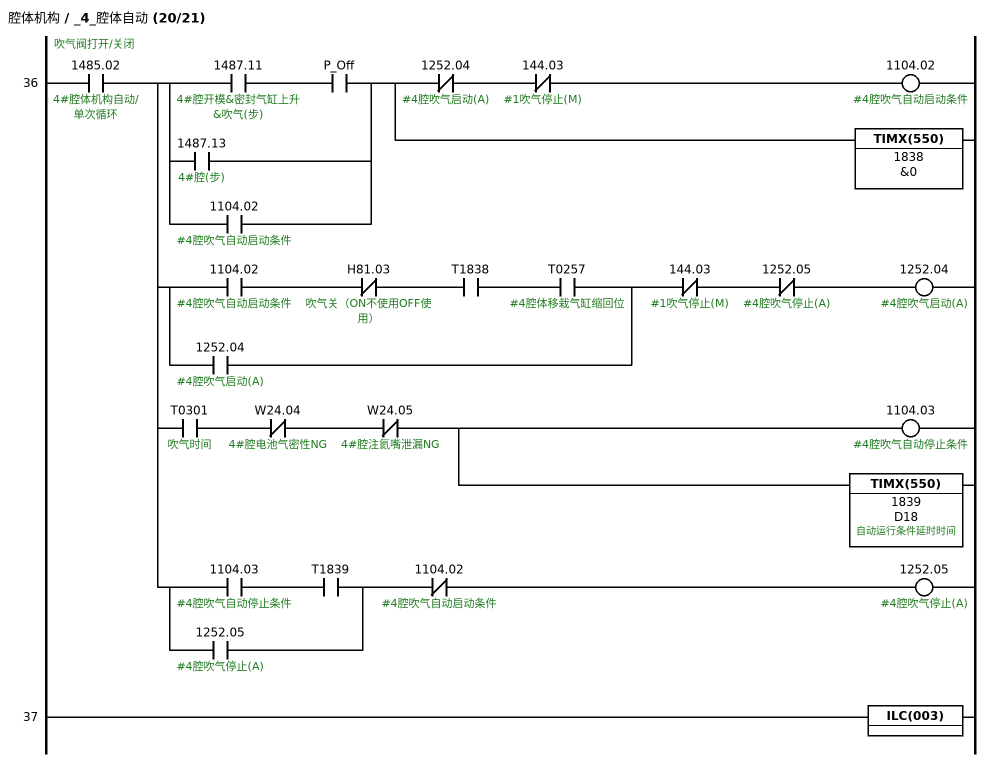
; [picture p360: 腔体机构 / _4_腔体自动, rungs 36-37]
; rung 36: 吹气阀打开/关闭
LD 1485.02  ; 4#腔体机构自动/单次循环
OUT TR0
LD 1487.11  ; 4#腔开模&密封气缸上升&吹气(步)
AND P_Off
OR 1487.13  ; 4#腔(步)
OR 1104.02  ; #4腔吹气自动启动条件
ANDLD
OUT TR1
ANDNOT 1252.04  ; #4腔吹气启动(A)
ANDNOT 144.03  ; #1吹气停止(M)
OUT 1104.02  ; #4腔吹气自动启动条件
LD TR1
TIMX(550) 1838 &0
LD TR0
LD 1104.02  ; #4腔吹气自动启动条件
ANDNOT H81.03  ; 吹气关（ON不使用OFF使用）
AND T1838
AND T0257  ; #4腔体移栽气缸缩回位
OR 1252.04  ; #4腔吹气启动(A)
ANDLD
ANDNOT 144.03  ; #1吹气停止(M)
ANDNOT 1252.05  ; #4腔吹气停止(A)
OUT 1252.04  ; #4腔吹气启动(A)
LD TR0
AND T0301  ; 吹气时间
ANDNOT W24.04  ; 4#腔电池气密性NG
ANDNOT W24.05  ; 4#腔注氦嘴泄漏NG
OUT 1104.03  ; #4腔吹气自动停止条件
TIMX(550) 1839 D18  ; 自动运行条件延时时间
LD TR0
LD 1104.03  ; #4腔吹气自动停止条件
AND T1839
OR 1252.05  ; #4腔吹气停止(A)
ANDLD
ANDNOT 1104.02  ; #4腔吹气自动启动条件
OUT 1252.05  ; #4腔吹气停止(A)
; rung 37
ILC(003)

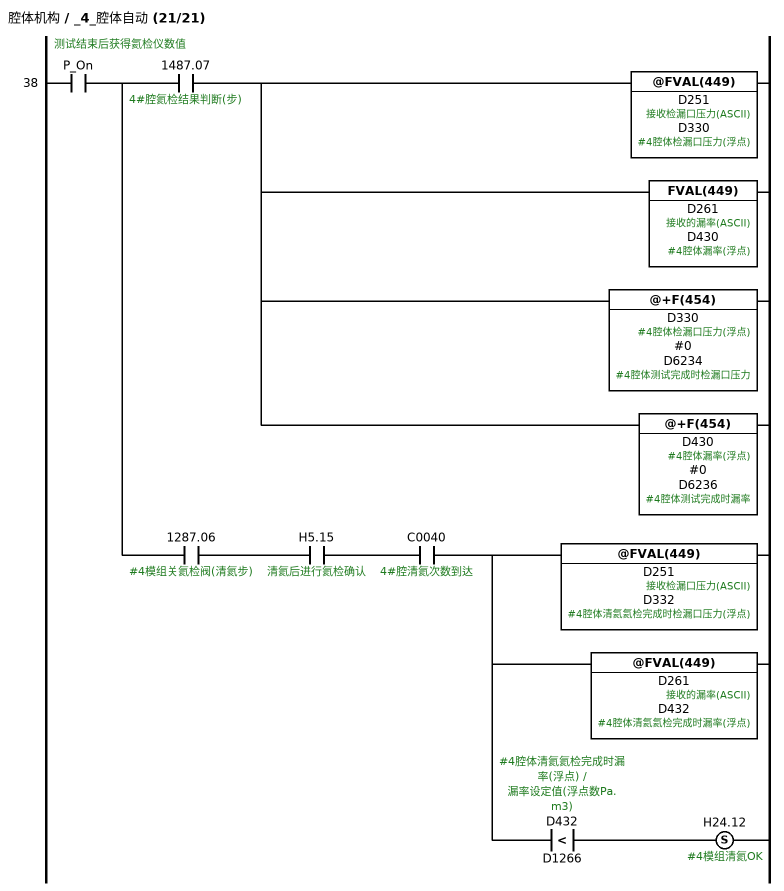
; rung 38: 测试结束后获得氦检仪数值
LD P_On
OUT TR0
AND 1487.07  ; 4#腔氦检结果判断(步)
@FVAL(449) D251 D330  ; 接收检漏口压力(ASCII), #4腔体检漏口压力(浮点)
FVAL(449) D261 D430  ; 接收的漏率(ASCII), #4腔体漏率(浮点)
@+F(454) D330 #0 D6234  ; #4腔体检漏口压力(浮点), #4腔体测试完成时检漏口压力
@+F(454) D430 #0 D6236  ; #4腔体漏率(浮点), #4腔体测试完成时漏率
LD TR0
AND 1287.06  ; #4模组关氦检阀(清氦步)
AND H5.15  ; 清氦后进行氦检确认
AND C0040  ; 4#腔清氦次数到达
@FVAL(449) D251 D332  ; 接收检漏口压力(ASCII), #4腔体清氦氦检完成时检漏口压力(浮点)
@FVAL(449) D261 D432  ; 接收的漏率(ASCII), #4腔体清氦氦检完成时漏率(浮点)
AND<F(331) D432 D1266  ; #4腔体清氦氦检完成时漏率(浮点), 漏率设定值(浮点数Pa.m3)
SET H24.12  ; #4模组清氦OK

### Section 外部输出

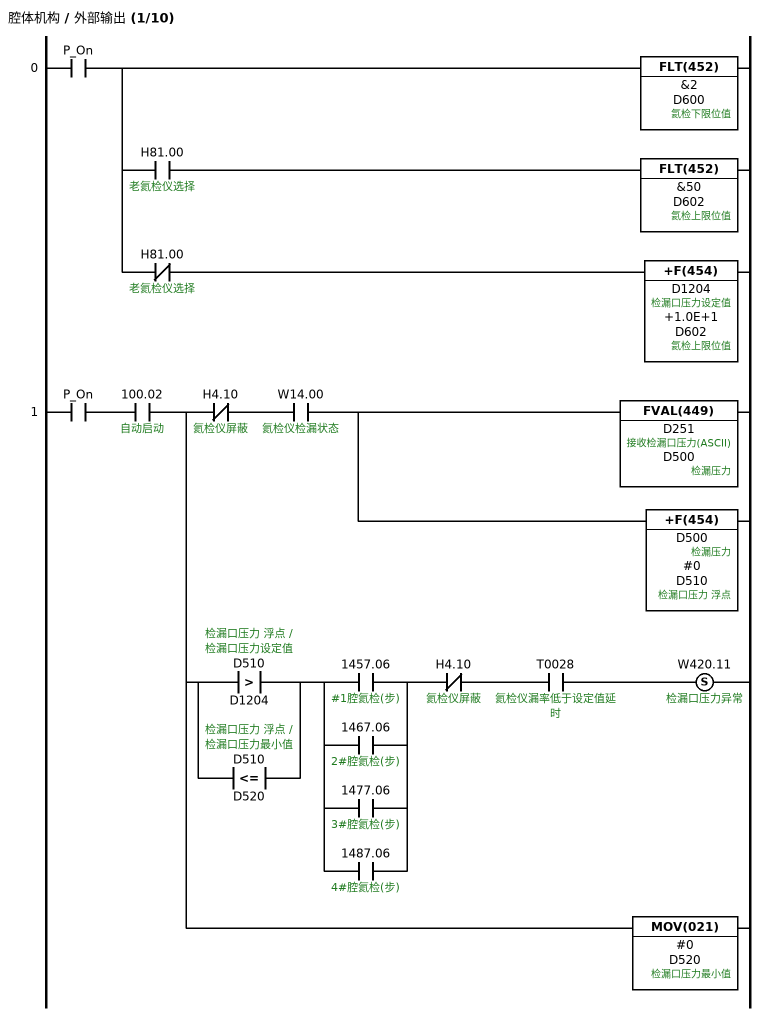
; rung 0
LD P_On
OUT TR0
FLT(452) &2 D600  ; 氦检下限位值
AND H81.00  ; 老氦检仪选择
FLT(452) &50 D602  ; 氦检上限位值
LD TR0
ANDNOT H81.00  ; 老氦检仪选择
+F(454) D1204 +1.0E+1 D602  ; 检漏口压力设定值, 氦检上限位值
; rung 1
LD P_On
AND 100.02  ; 自动启动
OUT TR0
ANDNOT H4.10  ; 氦检仪屏蔽
AND W14.00  ; 氦检仪检漏状态
FVAL(449) D251 D500  ; 接收检漏口压力(ASCII), 检漏压力
+F(454) D500 #0 D510  ; 检漏压力, 检漏口压力 浮点
LD TR0
LD>F(333) D510 D1204  ; 检漏口压力 浮点, 检漏口压力设定值
OR<=F(332) D510 D520  ; 检漏口压力 浮点, 检漏口压力最小值
ANDLD
LD 1457.06  ; #1腔氦检(步)
OR 1467.06  ; 2#腔氦检(步)
OR 1477.06  ; 3#腔氦检(步)
OR 1487.06  ; 4#腔氦检(步)
ANDLD
ANDNOT H4.10  ; 氦检仪屏蔽
AND T0028  ; 氦检仪漏率低于设定值延时
SET W420.11  ; 检漏口压力异常
LD TR0
MOV(021) #0 D520  ; 检漏口压力最小值

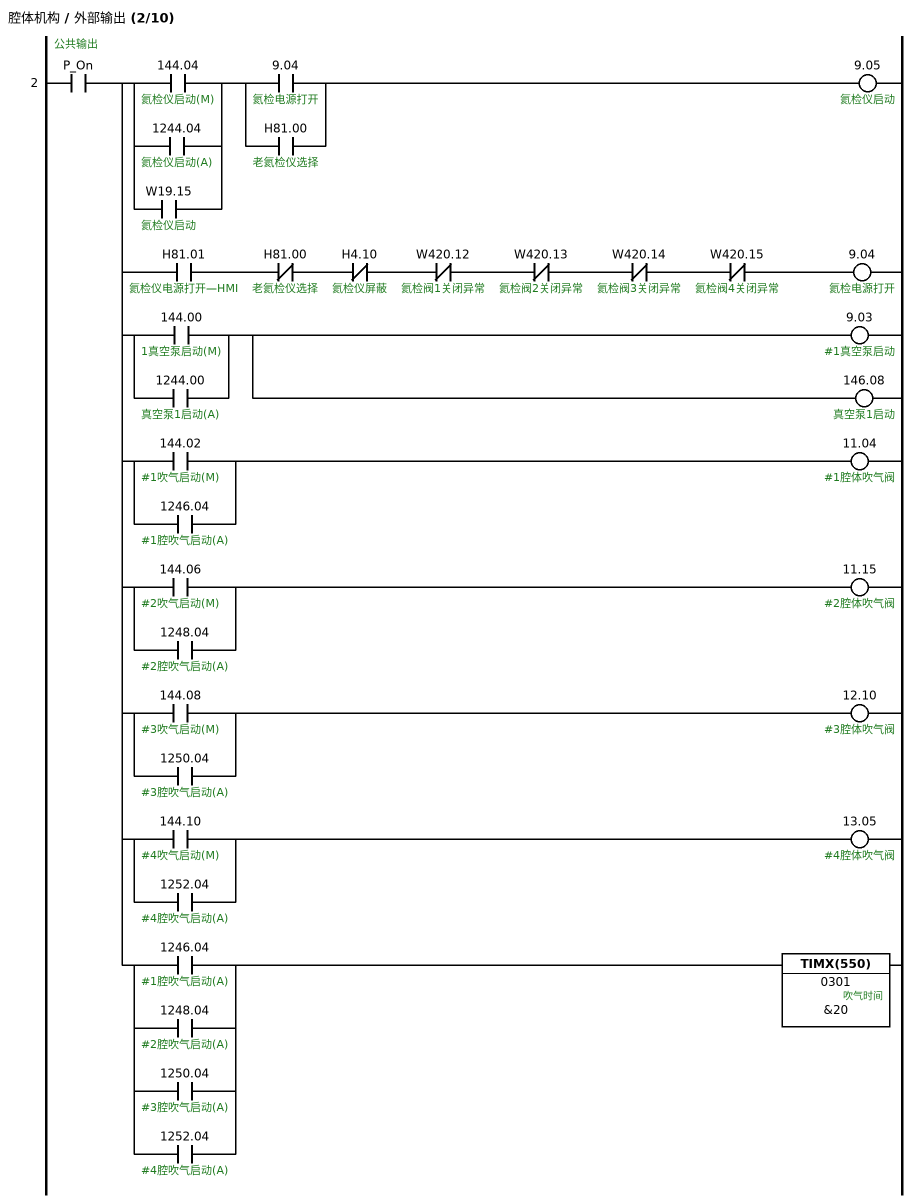
; rung 2: 公共输出
LD P_On
OUT TR0
LD 144.04  ; 氦检仪启动(M)
OR 1244.04  ; 氦检仪启动(A)
OR W19.15  ; 氦检仪启动
ANDLD
LD 9.04  ; 氦检电源打开
OR H81.00  ; 老氦检仪选择
ANDLD
OUT 9.05  ; 氦检仪启动
LD TR0
AND H81.01  ; 氦检仪电源打开—HMI
ANDNOT H81.00  ; 老氦检仪选择
ANDNOT H4.10  ; 氦检仪屏蔽
ANDNOT W420.12  ; 氦检阀1关闭异常
ANDNOT W420.13  ; 氦检阀2关闭异常
ANDNOT W420.14  ; 氦检阀3关闭异常
ANDNOT W420.15  ; 氦检阀4关闭异常
OUT 9.04  ; 氦检电源打开
LD TR0
LD 144.00  ; 1真空泵启动(M)
OR 1244.00  ; 真空泵1启动(A)
ANDLD
OUT 9.03  ; #1真空泵启动
OUT 146.08  ; 真空泵1启动
LD TR0
LD 144.02  ; #1吹气启动(M)
OR 1246.04  ; #1腔吹气启动(A)
ANDLD
OUT 11.04  ; #1腔体吹气阀
LD TR0
LD 144.06  ; #2吹气启动(M)
OR 1248.04  ; #2腔吹气启动(A)
ANDLD
OUT 11.15  ; #2腔体吹气阀
LD TR0
LD 144.08  ; #3吹气启动(M)
OR 1250.04  ; #3腔吹气启动(A)
ANDLD
OUT 12.10  ; #3腔体吹气阀
LD TR0
LD 144.10  ; #4吹气启动(M)
OR 1252.04  ; #4腔吹气启动(A)
ANDLD
OUT 13.05  ; #4腔体吹气阀
LD TR0
LD 1246.04  ; #1腔吹气启动(A)
OR 1248.04  ; #2腔吹气启动(A)
OR 1250.04  ; #3腔吹气启动(A)
OR 1252.04  ; #4腔吹气启动(A)
ANDLD
TIMX(550) 0301 &20  ; 吹气时间

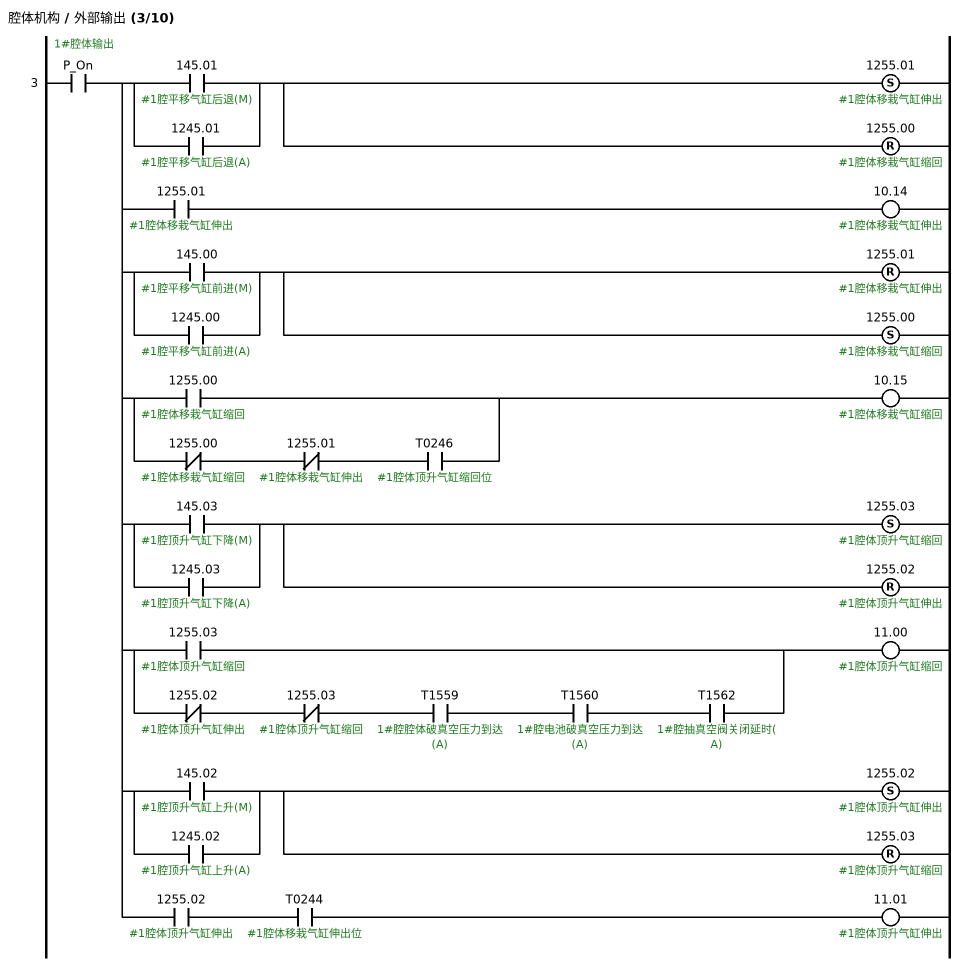
; rung 3: 1#腔体输出
LD P_On
OUT TR0
LD 145.01  ; #1腔平移气缸后退(M)
OR 1245.01  ; #1腔平移气缸后退(A)
ANDLD
SET 1255.01  ; #1腔体移栽气缸伸出
RSET 1255.00  ; #1腔体移栽气缸缩回
LD TR0
AND 1255.01  ; #1腔体移栽气缸伸出
OUT 10.14  ; #1腔体移栽气缸伸出
LD TR0
LD 145.00  ; #1腔平移气缸前进(M)
OR 1245.00  ; #1腔平移气缸前进(A)
ANDLD
RSET 1255.01  ; #1腔体移栽气缸伸出
SET 1255.00  ; #1腔体移栽气缸缩回
LD TR0
LD 1255.00  ; #1腔体移栽气缸缩回
LDNOT 1255.00  ; #1腔体移栽气缸缩回
ANDNOT 1255.01  ; #1腔体移栽气缸伸出
AND T0246  ; #1腔体顶升气缸缩回位
ORLD
ANDLD
OUT 10.15  ; #1腔体移栽气缸缩回
LD TR0
LD 145.03  ; #1腔顶升气缸下降(M)
OR 1245.03  ; #1腔顶升气缸下降(A)
ANDLD
SET 1255.03  ; #1腔体顶升气缸缩回
RSET 1255.02  ; #1腔体顶升气缸伸出
LD TR0
LD 1255.03  ; #1腔体顶升气缸缩回
LDNOT 1255.02  ; #1腔体顶升气缸伸出
ANDNOT 1255.03  ; #1腔体顶升气缸缩回
AND T1559  ; 1#腔腔体破真空压力到达(A)
AND T1560  ; 1#腔电池破真空压力到达(A)
AND T1562  ; 1#腔抽真空阀关闭延时(A)
ORLD
ANDLD
OUT 11.00  ; #1腔体顶升气缸缩回
LD TR0
LD 145.02  ; #1腔顶升气缸上升(M)
OR 1245.02  ; #1腔顶升气缸上升(A)
ANDLD
SET 1255.02  ; #1腔体顶升气缸伸出
RSET 1255.03  ; #1腔体顶升气缸缩回
LD TR0
AND 1255.02  ; #1腔体顶升气缸伸出
AND T0244  ; #1腔体移栽气缸伸出位
OUT 11.01  ; #1腔体顶升气缸伸出

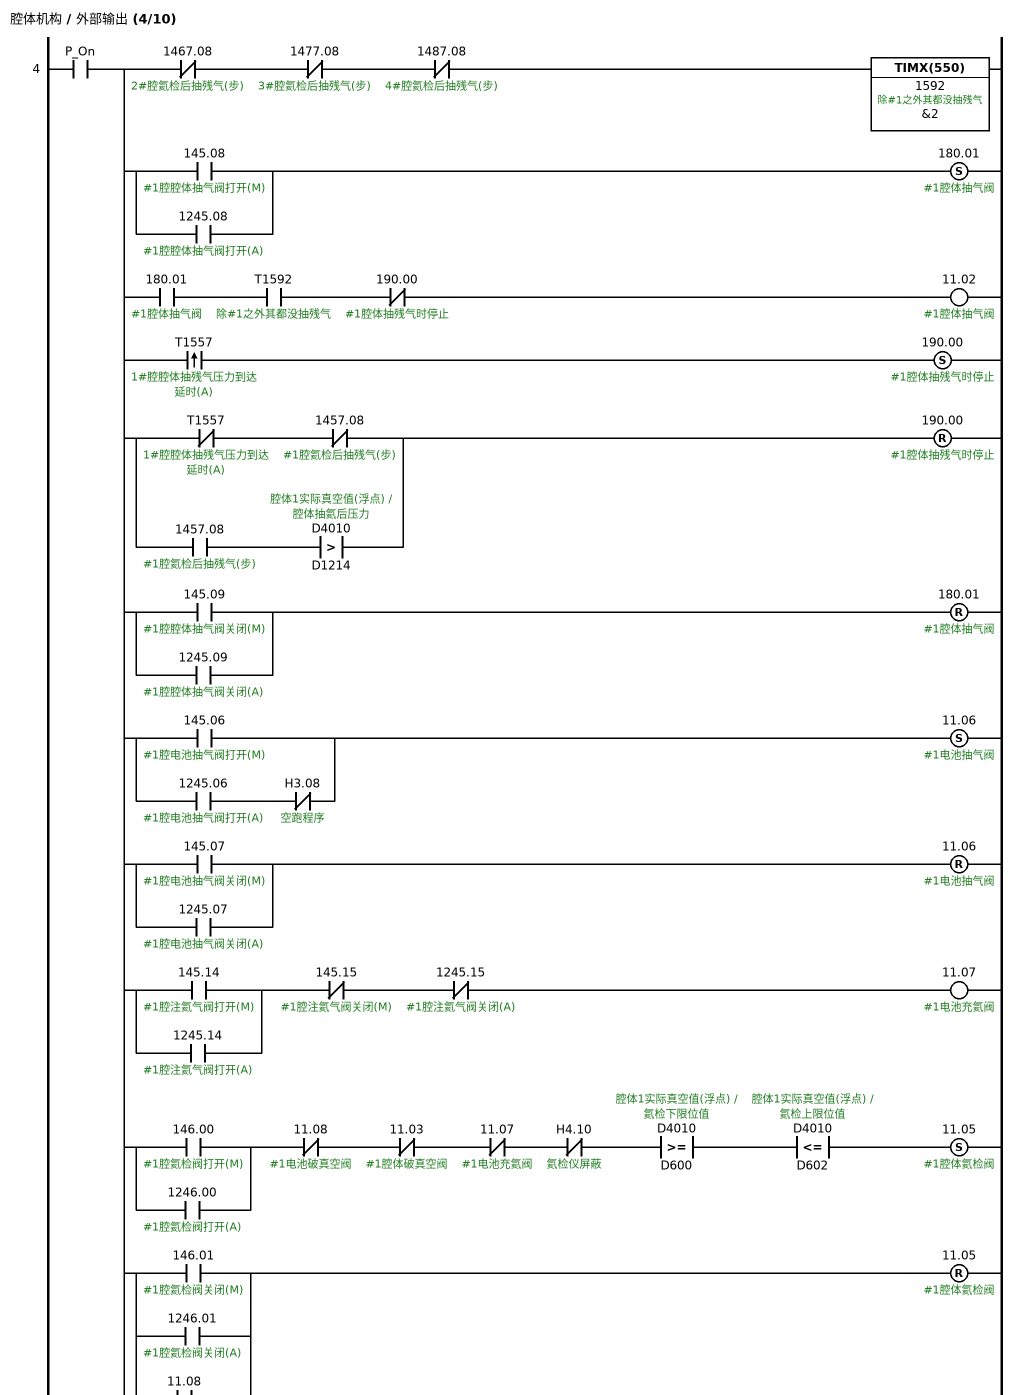

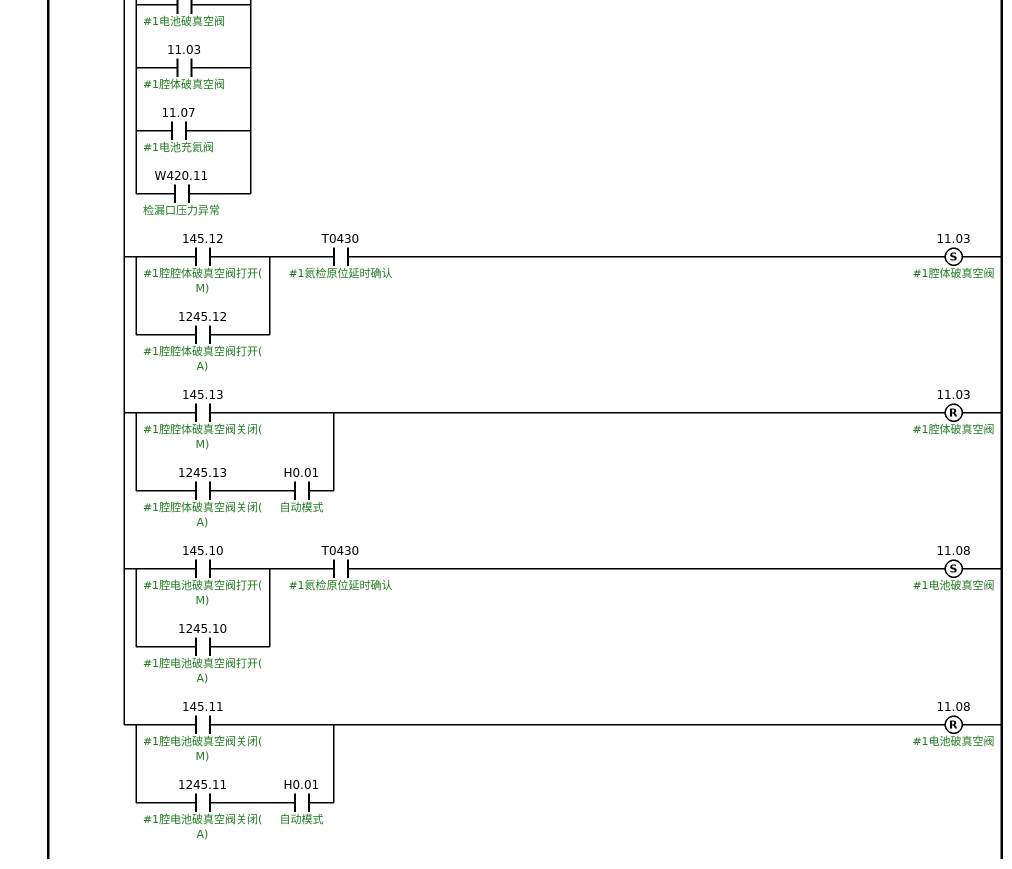
; rung 4
LD P_On
OUT TR0
ANDNOT 1467.08  ; 2#腔氦检后抽残气(步)
ANDNOT 1477.08  ; 3#腔氦检后抽残气(步)
ANDNOT 1487.08  ; 4#腔氦检后抽残气(步)
TIMX(550) 1592 &2  ; 除#1之外其都没抽残气
LD TR0
LD 145.08  ; #1腔腔体抽气阀打开(M)
OR 1245.08  ; #1腔腔体抽气阀打开(A)
ANDLD
SET 180.01  ; #1腔体抽气阀
LD TR0
AND 180.01  ; #1腔体抽气阀
AND T1592  ; 除#1之外其都没抽残气
ANDNOT 190.00  ; #1腔体抽残气时停止
OUT 11.02  ; #1腔体抽气阀
LD TR0
@AND T1557  ; 1#腔腔体抽残气压力到达延时(A)
SET 190.00  ; #1腔体抽残气时停止
LD TR0
LDNOT T1557  ; 1#腔腔体抽残气压力到达延时(A)
ANDNOT 1457.08  ; #1腔氦检后抽残气(步)
LD 1457.08  ; #1腔氦检后抽残气(步)
AND>F(333) D4010 D1214  ; 腔体1实际真空值(浮点), 腔体抽氦后压力
ORLD
ANDLD
RSET 190.00  ; #1腔体抽残气时停止
LD TR0
LD 145.09  ; #1腔腔体抽气阀关闭(M)
OR 1245.09  ; #1腔腔体抽气阀关闭(A)
ANDLD
RSET 180.01  ; #1腔体抽气阀
LD TR0
LD 145.06  ; #1腔电池抽气阀打开(M)
LD 1245.06  ; #1腔电池抽气阀打开(A)
ANDNOT H3.08  ; 空跑程序
ORLD
ANDLD
SET 11.06  ; #1电池抽气阀
LD TR0
LD 145.07  ; #1腔电池抽气阀关闭(M)
OR 1245.07  ; #1腔电池抽气阀关闭(A)
ANDLD
RSET 11.06  ; #1电池抽气阀
LD TR0
LD 145.14  ; #1腔注氦气阀打开(M)
OR 1245.14  ; #1腔注氦气阀打开(A)
ANDLD
ANDNOT 145.15  ; #1腔注氦气阀关闭(M)
ANDNOT 1245.15  ; #1腔注氦气阀关闭(A)
OUT 11.07  ; #1电池充氦阀
LD TR0
LD 146.00  ; #1腔氦检阀打开(M)
OR 1246.00  ; #1腔氦检阀打开(A)
ANDLD
ANDNOT 11.08  ; #1电池破真空阀
ANDNOT 11.03  ; #1腔体破真空阀
ANDNOT 11.07  ; #1电池充氦阀
ANDNOT H4.10  ; 氦检仪屏蔽
AND>=F(334) D4010 D600  ; 腔体1实际真空值(浮点), 氦检下限位值
AND<=F(332) D4010 D602  ; 腔体1实际真空值(浮点), 氦检上限位值
SET 11.05  ; #1腔体氦检阀
LD TR0
LD 146.01  ; #1腔氦检阀关闭(M)
OR 1246.01  ; #1腔氦检阀关闭(A)
OR 11.08  ; #1电池破真空阀
OR 11.03  ; #1腔体破真空阀
OR 11.07  ; #1电池充氦阀
OR W420.11  ; 检漏口压力异常
ANDLD
RSET 11.05  ; #1腔体氦检阀
LD TR0
LD 145.12  ; #1腔腔体破真空阀打开(M)
OR 1245.12  ; #1腔腔体破真空阀打开(A)
ANDLD
AND T0430  ; #1氦检原位延时确认
SET 11.03  ; #1腔体破真空阀
LD TR0
LD 145.13  ; #1腔腔体破真空阀关闭(M)
LD 1245.13  ; #1腔腔体破真空阀关闭(A)
AND H0.01  ; 自动模式
ORLD
ANDLD
RSET 11.03  ; #1腔体破真空阀
LD TR0
LD 145.10  ; #1腔电池破真空阀打开(M)
OR 1245.10  ; #1腔电池破真空阀打开(A)
ANDLD
AND T0430  ; #1氦检原位延时确认
SET 11.08  ; #1电池破真空阀
LD TR0
LD 145.11  ; #1腔电池破真空阀关闭(M)
LD 1245.11  ; #1腔电池破真空阀关闭(A)
AND H0.01  ; 自动模式
ORLD
ANDLD
RSET 11.08  ; #1电池破真空阀

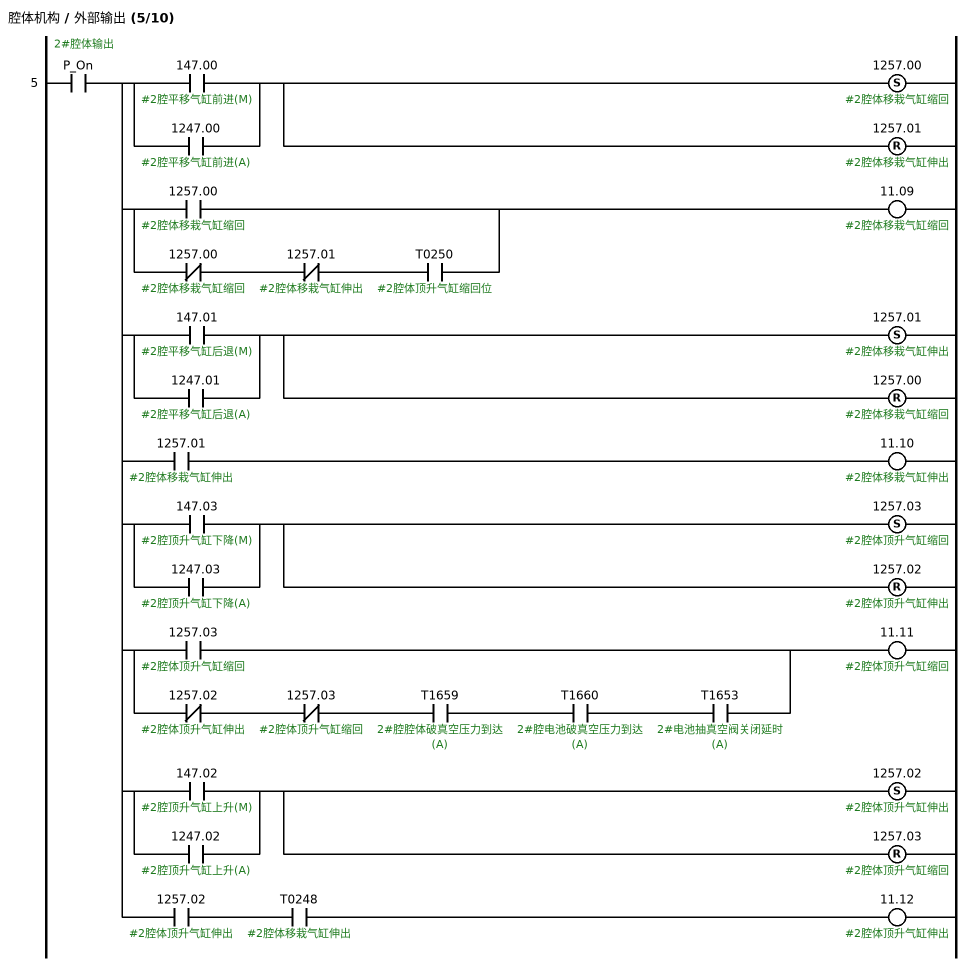
; rung 5: 2#腔体输出
LD P_On
OUT TR0
LD 147.00  ; #2腔平移气缸前进(M)
OR 1247.00  ; #2腔平移气缸前进(A)
ANDLD
SET 1257.00  ; #2腔体移栽气缸缩回
RSET 1257.01  ; #2腔体移栽气缸伸出
LD TR0
LD 1257.00  ; #2腔体移栽气缸缩回
LDNOT 1257.00  ; #2腔体移栽气缸缩回
ANDNOT 1257.01  ; #2腔体移栽气缸伸出
AND T0250  ; #2腔体顶升气缸缩回位
ORLD
ANDLD
OUT 11.09  ; #2腔体移栽气缸缩回
LD TR0
LD 147.01  ; #2腔平移气缸后退(M)
OR 1247.01  ; #2腔平移气缸后退(A)
ANDLD
SET 1257.01  ; #2腔体移栽气缸伸出
RSET 1257.00  ; #2腔体移栽气缸缩回
LD TR0
AND 1257.01  ; #2腔体移栽气缸伸出
OUT 11.10  ; #2腔体移栽气缸伸出
LD TR0
LD 147.03  ; #2腔顶升气缸下降(M)
OR 1247.03  ; #2腔顶升气缸下降(A)
ANDLD
SET 1257.03  ; #2腔体顶升气缸缩回
RSET 1257.02  ; #2腔体顶升气缸伸出
LD TR0
LD 1257.03  ; #2腔体顶升气缸缩回
LDNOT 1257.02  ; #2腔体顶升气缸伸出
ANDNOT 1257.03  ; #2腔体顶升气缸缩回
AND T1659  ; 2#腔腔体破真空压力到达(A)
AND T1660  ; 2#腔电池破真空压力到达(A)
AND T1653  ; 2#电池抽真空阀关闭延时(A)
ORLD
ANDLD
OUT 11.11  ; #2腔体顶升气缸缩回
LD TR0
LD 147.02  ; #2腔顶升气缸上升(M)
OR 1247.02  ; #2腔顶升气缸上升(A)
ANDLD
SET 1257.02  ; #2腔体顶升气缸伸出
RSET 1257.03  ; #2腔体顶升气缸缩回
LD TR0
AND 1257.02  ; #2腔体顶升气缸伸出
AND T0248  ; #2腔体移栽气缸伸出
OUT 11.12  ; #2腔体顶升气缸伸出

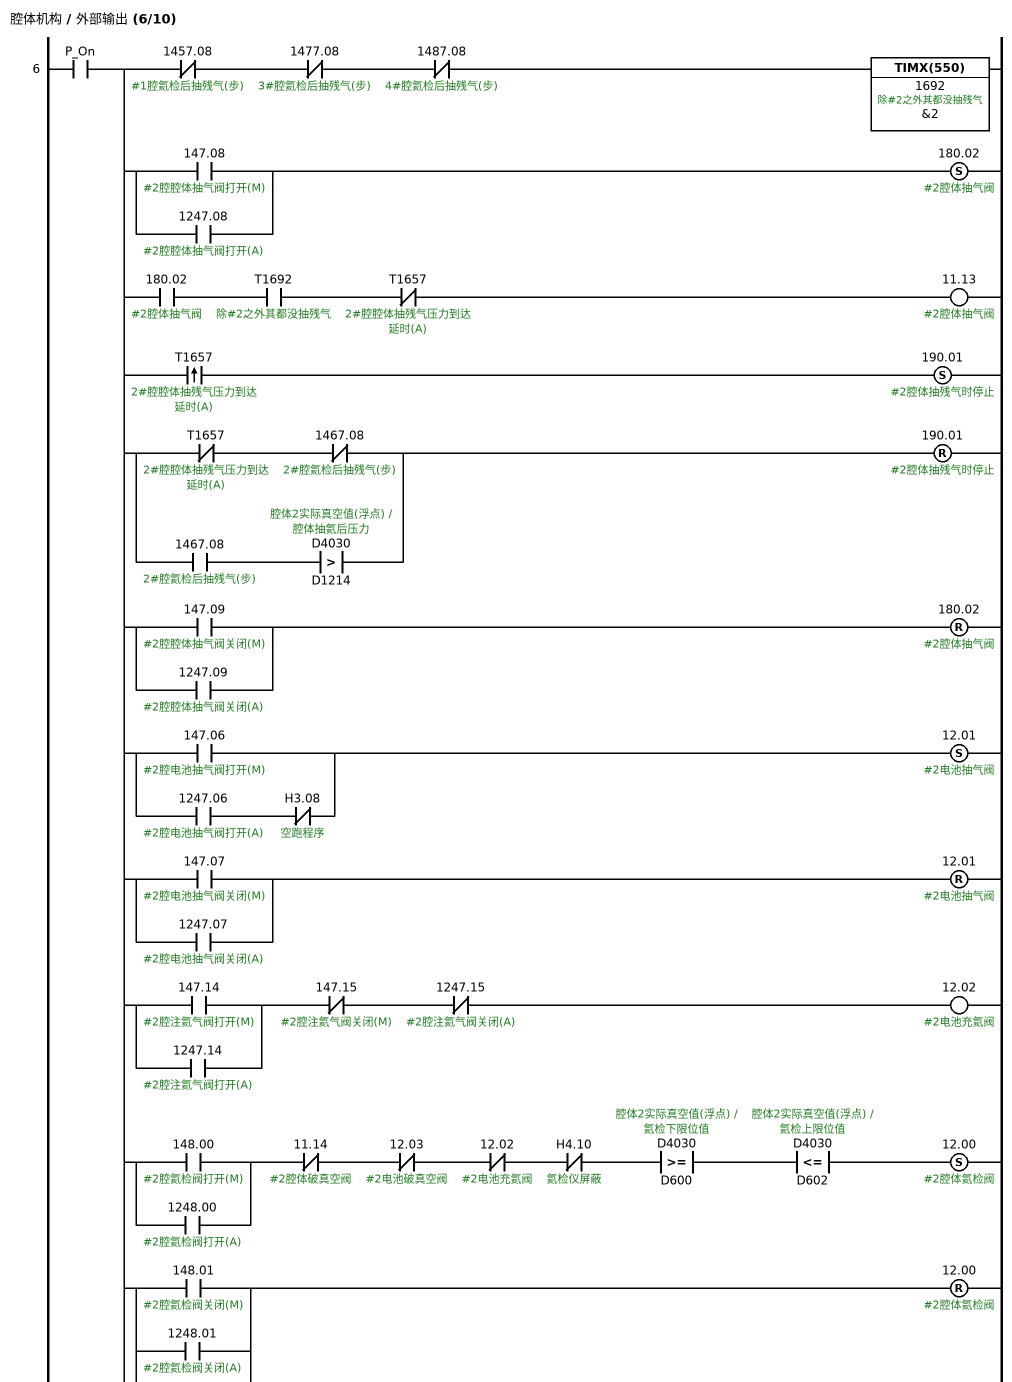

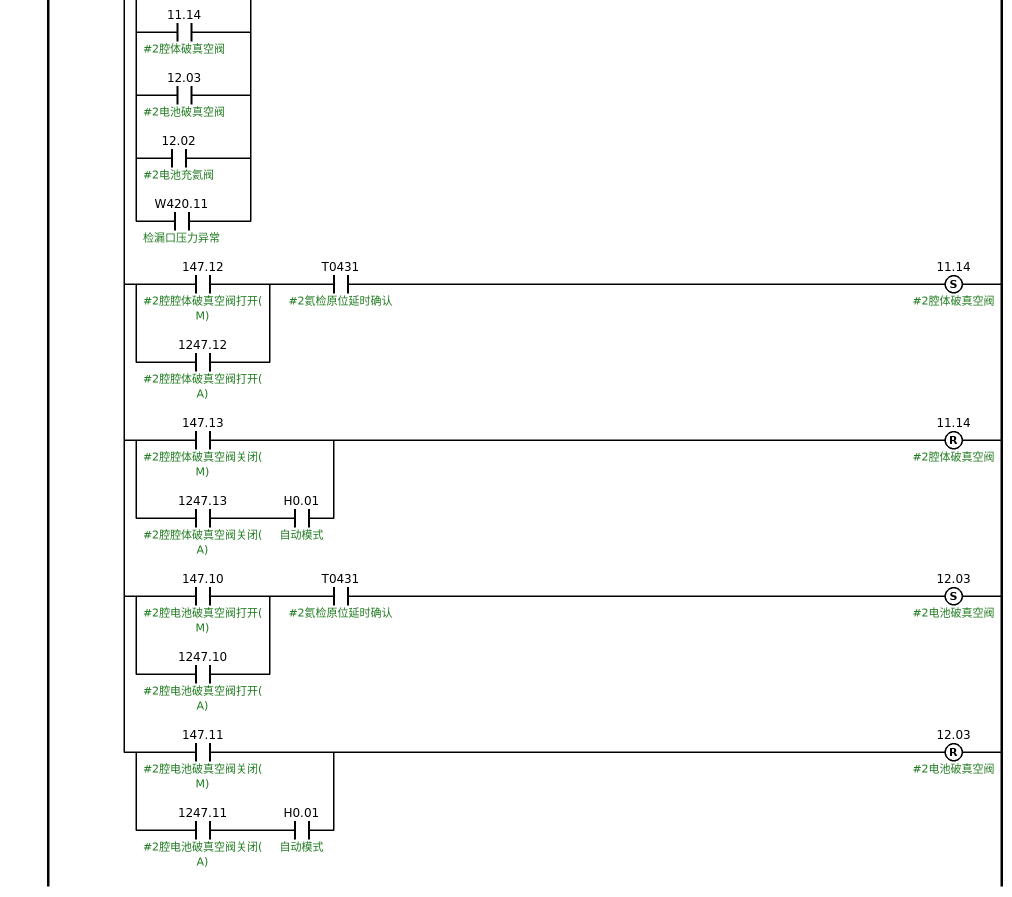
; rung 6
LD P_On
OUT TR0
ANDNOT 1457.08  ; #1腔氦检后抽残气(步)
ANDNOT 1477.08  ; 3#腔氦检后抽残气(步)
ANDNOT 1487.08  ; 4#腔氦检后抽残气(步)
TIMX(550) 1692 &2  ; 除#2之外其都没抽残气
LD TR0
LD 147.08  ; #2腔腔体抽气阀打开(M)
OR 1247.08  ; #2腔腔体抽气阀打开(A)
ANDLD
SET 180.02  ; #2腔体抽气阀
LD TR0
AND 180.02  ; #2腔体抽气阀
AND T1692  ; 除#2之外其都没抽残气
ANDNOT T1657  ; 2#腔腔体抽残气压力到达延时(A)
OUT 11.13  ; #2腔体抽气阀
LD TR0
@AND T1657  ; 2#腔腔体抽残气压力到达延时(A)
SET 190.01  ; #2腔体抽残气时停止
LD TR0
LDNOT T1657  ; 2#腔腔体抽残气压力到达延时(A)
ANDNOT 1467.08  ; 2#腔氦检后抽残气(步)
LD 1467.08  ; 2#腔氦检后抽残气(步)
AND>F(333) D4030 D1214  ; 腔体2实际真空值(浮点), 腔体抽氦后压力
ORLD
ANDLD
RSET 190.01  ; #2腔体抽残气时停止
LD TR0
LD 147.09  ; #2腔腔体抽气阀关闭(M)
OR 1247.09  ; #2腔腔体抽气阀关闭(A)
ANDLD
RSET 180.02  ; #2腔体抽气阀
LD TR0
LD 147.06  ; #2腔电池抽气阀打开(M)
LD 1247.06  ; #2腔电池抽气阀打开(A)
ANDNOT H3.08  ; 空跑程序
ORLD
ANDLD
SET 12.01  ; #2电池抽气阀
LD TR0
LD 147.07  ; #2腔电池抽气阀关闭(M)
OR 1247.07  ; #2腔电池抽气阀关闭(A)
ANDLD
RSET 12.01  ; #2电池抽气阀
LD TR0
LD 147.14  ; #2腔注氦气阀打开(M)
OR 1247.14  ; #2腔注氦气阀打开(A)
ANDLD
ANDNOT 147.15  ; #2腔注氦气阀关闭(M)
ANDNOT 1247.15  ; #2腔注氦气阀关闭(A)
OUT 12.02  ; #2电池充氦阀
LD TR0
LD 148.00  ; #2腔氦检阀打开(M)
OR 1248.00  ; #2腔氦检阀打开(A)
ANDLD
ANDNOT 11.14  ; #2腔体破真空阀
ANDNOT 12.03  ; #2电池破真空阀
ANDNOT 12.02  ; #2电池充氦阀
ANDNOT H4.10  ; 氦检仪屏蔽
AND>=F(334) D4030 D600  ; 腔体2实际真空值(浮点), 氦检下限位值
AND<=F(332) D4030 D602  ; 腔体2实际真空值(浮点), 氦检上限位值
SET 12.00  ; #2腔体氦检阀
LD TR0
LD 148.01  ; #2腔氦检阀关闭(M)
OR 1248.01  ; #2腔氦检阀关闭(A)
OR 11.14  ; #2腔体破真空阀
OR 12.03  ; #2电池破真空阀
OR 12.02  ; #2电池充氦阀
OR W420.11  ; 检漏口压力异常
ANDLD
RSET 12.00  ; #2腔体氦检阀
LD TR0
LD 147.12  ; #2腔腔体破真空阀打开(M)
OR 1247.12  ; #2腔腔体破真空阀打开(A)
ANDLD
AND T0431  ; #2氦检原位延时确认
SET 11.14  ; #2腔体破真空阀
LD TR0
LD 147.13  ; #2腔腔体破真空阀关闭(M)
LD 1247.13  ; #2腔腔体破真空阀关闭(A)
AND H0.01  ; 自动模式
ORLD
ANDLD
RSET 11.14  ; #2腔体破真空阀
LD TR0
LD 147.10  ; #2腔电池破真空阀打开(M)
OR 1247.10  ; #2腔电池破真空阀打开(A)
ANDLD
AND T0431  ; #2氦检原位延时确认
SET 12.03  ; #2电池破真空阀
LD TR0
LD 147.11  ; #2腔电池破真空阀关闭(M)
LD 1247.11  ; #2腔电池破真空阀关闭(A)
AND H0.01  ; 自动模式
ORLD
ANDLD
RSET 12.03  ; #2电池破真空阀

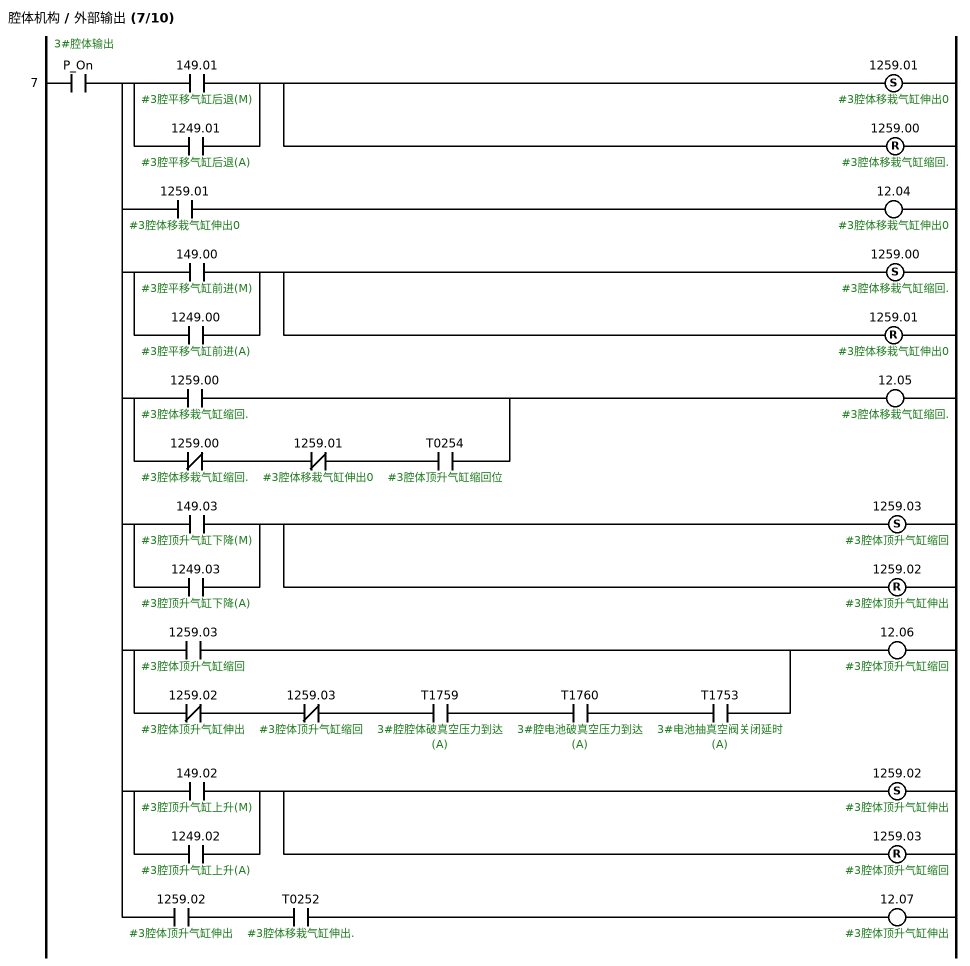
; rung 7: 3#腔体输出
LD P_On
OUT TR0
LD 149.01  ; #3腔平移气缸后退(M)
OR 1249.01  ; #3腔平移气缸后退(A)
ANDLD
SET 1259.01  ; #3腔体移栽气缸伸出0
RSET 1259.00  ; #3腔体移栽气缸缩回.
LD TR0
AND 1259.01  ; #3腔体移栽气缸伸出0
OUT 12.04  ; #3腔体移栽气缸伸出0
LD TR0
LD 149.00  ; #3腔平移气缸前进(M)
OR 1249.00  ; #3腔平移气缸前进(A)
ANDLD
SET 1259.00  ; #3腔体移栽气缸缩回.
RSET 1259.01  ; #3腔体移栽气缸伸出0
LD TR0
LD 1259.00  ; #3腔体移栽气缸缩回.
LDNOT 1259.00  ; #3腔体移栽气缸缩回.
ANDNOT 1259.01  ; #3腔体移栽气缸伸出0
AND T0254  ; #3腔体顶升气缸缩回位
ORLD
ANDLD
OUT 12.05  ; #3腔体移栽气缸缩回.
LD TR0
LD 149.03  ; #3腔顶升气缸下降(M)
OR 1249.03  ; #3腔顶升气缸下降(A)
ANDLD
SET 1259.03  ; #3腔体顶升气缸缩回
RSET 1259.02  ; #3腔体顶升气缸伸出
LD TR0
LD 1259.03  ; #3腔体顶升气缸缩回
LDNOT 1259.02  ; #3腔体顶升气缸伸出
ANDNOT 1259.03  ; #3腔体顶升气缸缩回
AND T1759  ; 3#腔腔体破真空压力到达(A)
AND T1760  ; 3#腔电池破真空压力到达(A)
AND T1753  ; 3#电池抽真空阀关闭延时(A)
ORLD
ANDLD
OUT 12.06  ; #3腔体顶升气缸缩回
LD TR0
LD 149.02  ; #3腔顶升气缸上升(M)
OR 1249.02  ; #3腔顶升气缸上升(A)
ANDLD
SET 1259.02  ; #3腔体顶升气缸伸出
RSET 1259.03  ; #3腔体顶升气缸缩回
LD TR0
AND 1259.02  ; #3腔体顶升气缸伸出
AND T0252  ; #3腔体移栽气缸伸出.
OUT 12.07  ; #3腔体顶升气缸伸出

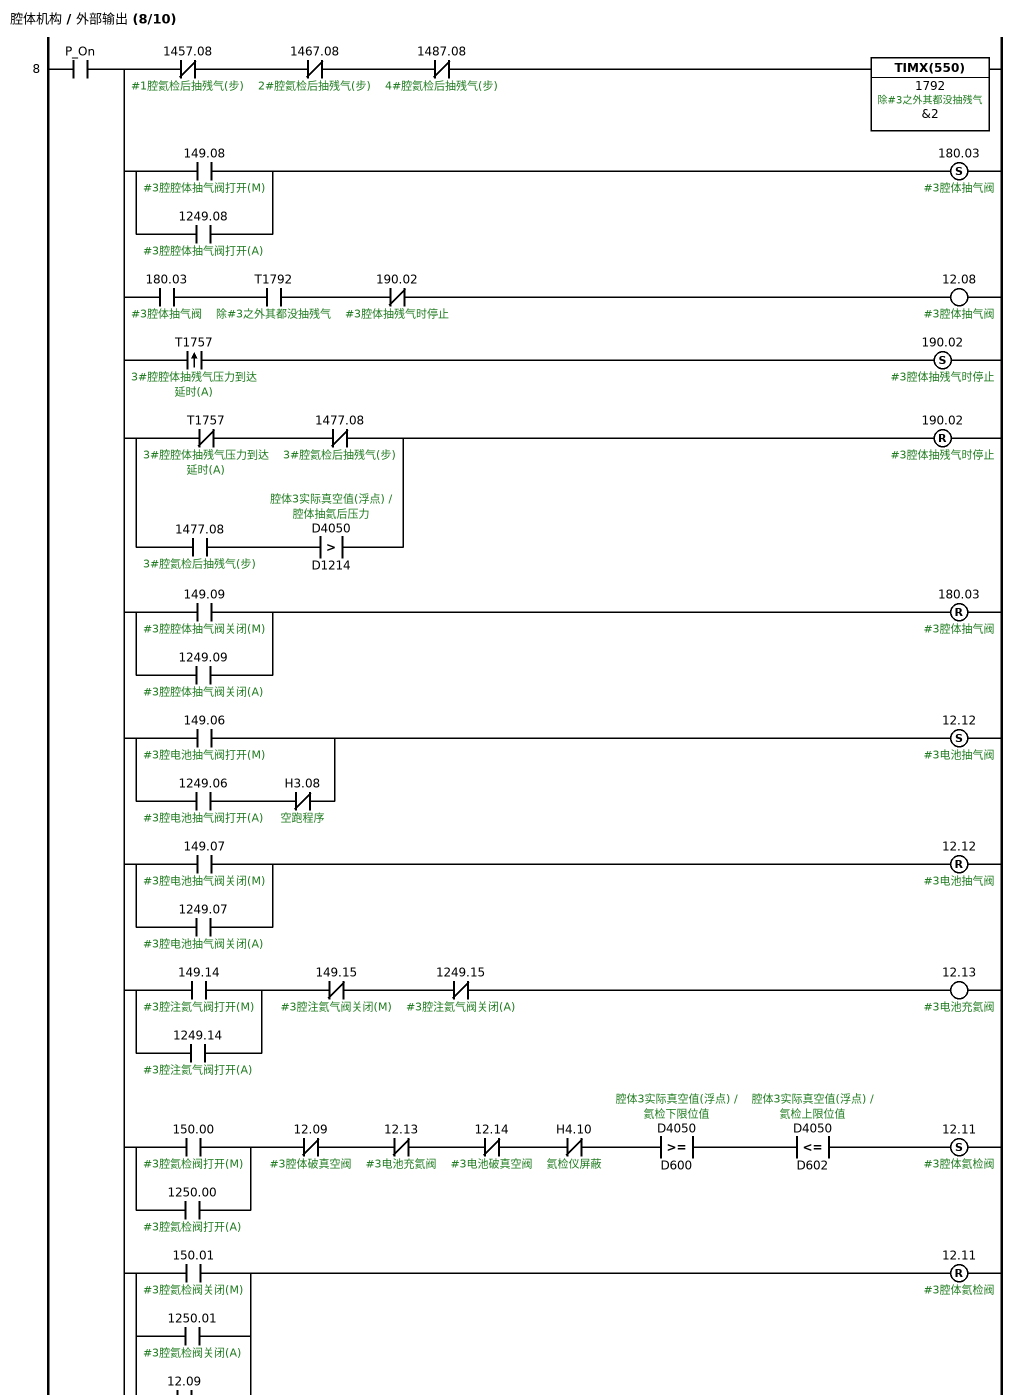

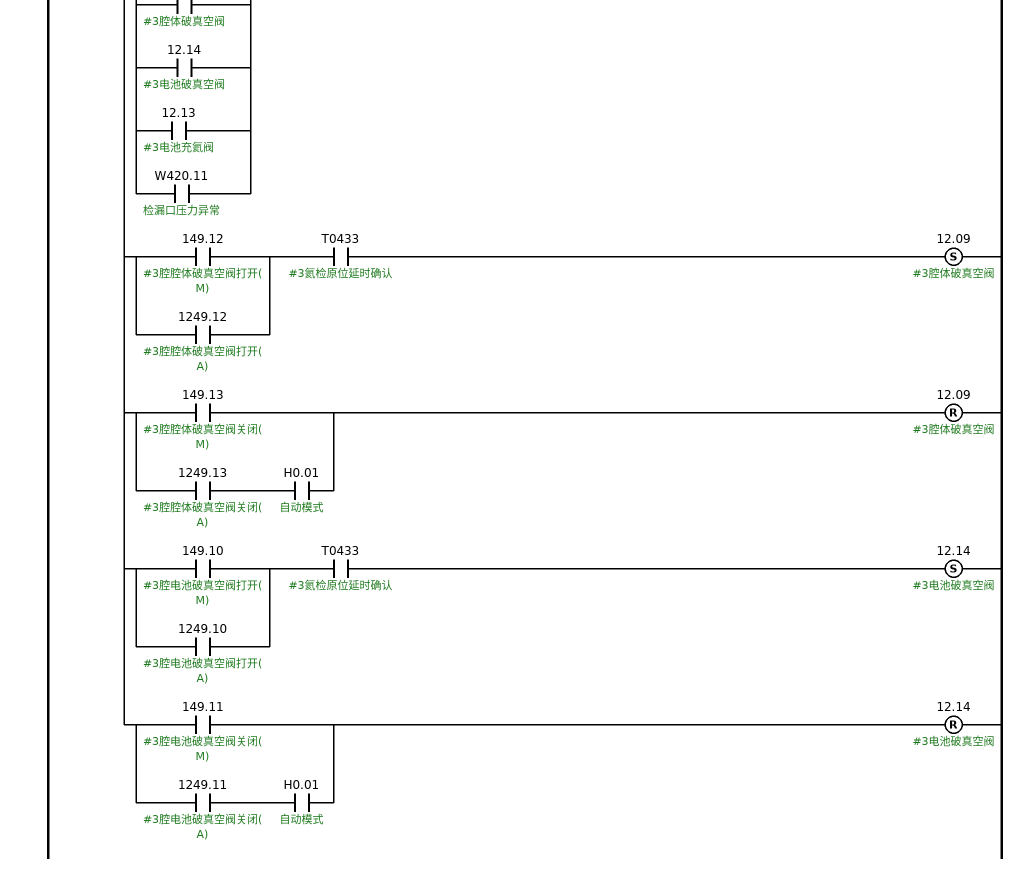
; rung 8
LD P_On
OUT TR0
ANDNOT 1457.08  ; #1腔氦检后抽残气(步)
ANDNOT 1467.08  ; 2#腔氦检后抽残气(步)
ANDNOT 1487.08  ; 4#腔氦检后抽残气(步)
TIMX(550) 1792 &2  ; 除#3之外其都没抽残气
LD TR0
LD 149.08  ; #3腔腔体抽气阀打开(M)
OR 1249.08  ; #3腔腔体抽气阀打开(A)
ANDLD
SET 180.03  ; #3腔体抽气阀
LD TR0
AND 180.03  ; #3腔体抽气阀
AND T1792  ; 除#3之外其都没抽残气
ANDNOT 190.02  ; #3腔体抽残气时停止
OUT 12.08  ; #3腔体抽气阀
LD TR0
@AND T1757  ; 3#腔腔体抽残气压力到达延时(A)
SET 190.02  ; #3腔体抽残气时停止
LD TR0
LDNOT T1757  ; 3#腔腔体抽残气压力到达延时(A)
ANDNOT 1477.08  ; 3#腔氦检后抽残气(步)
LD 1477.08  ; 3#腔氦检后抽残气(步)
AND>F(333) D4050 D1214  ; 腔体3实际真空值(浮点), 腔体抽氦后压力
ORLD
ANDLD
RSET 190.02  ; #3腔体抽残气时停止
LD TR0
LD 149.09  ; #3腔腔体抽气阀关闭(M)
OR 1249.09  ; #3腔腔体抽气阀关闭(A)
ANDLD
RSET 180.03  ; #3腔体抽气阀
LD TR0
LD 149.06  ; #3腔电池抽气阀打开(M)
LD 1249.06  ; #3腔电池抽气阀打开(A)
ANDNOT H3.08  ; 空跑程序
ORLD
ANDLD
SET 12.12  ; #3电池抽气阀
LD TR0
LD 149.07  ; #3腔电池抽气阀关闭(M)
OR 1249.07  ; #3腔电池抽气阀关闭(A)
ANDLD
RSET 12.12  ; #3电池抽气阀
LD TR0
LD 149.14  ; #3腔注氦气阀打开(M)
OR 1249.14  ; #3腔注氦气阀打开(A)
ANDLD
ANDNOT 149.15  ; #3腔注氦气阀关闭(M)
ANDNOT 1249.15  ; #3腔注氦气阀关闭(A)
OUT 12.13  ; #3电池充氦阀
LD TR0
LD 150.00  ; #3腔氦检阀打开(M)
OR 1250.00  ; #3腔氦检阀打开(A)
ANDLD
ANDNOT 12.09  ; #3腔体破真空阀
ANDNOT 12.13  ; #3电池充氦阀
ANDNOT 12.14  ; #3电池破真空阀
ANDNOT H4.10  ; 氦检仪屏蔽
AND>=F(334) D4050 D600  ; 腔体3实际真空值(浮点), 氦检下限位值
AND<=F(332) D4050 D602  ; 腔体3实际真空值(浮点), 氦检上限位值
SET 12.11  ; #3腔体氦检阀
LD TR0
LD 150.01  ; #3腔氦检阀关闭(M)
OR 1250.01  ; #3腔氦检阀关闭(A)
OR 12.09  ; #3腔体破真空阀
OR 12.14  ; #3电池破真空阀
OR 12.13  ; #3电池充氦阀
OR W420.11  ; 检漏口压力异常
ANDLD
RSET 12.11  ; #3腔体氦检阀
LD TR0
LD 149.12  ; #3腔腔体破真空阀打开(M)
OR 1249.12  ; #3腔腔体破真空阀打开(A)
ANDLD
AND T0433  ; #3氦检原位延时确认
SET 12.09  ; #3腔体破真空阀
LD TR0
LD 149.13  ; #3腔腔体破真空阀关闭(M)
LD 1249.13  ; #3腔腔体破真空阀关闭(A)
AND H0.01  ; 自动模式
ORLD
ANDLD
RSET 12.09  ; #3腔体破真空阀
LD TR0
LD 149.10  ; #3腔电池破真空阀打开(M)
OR 1249.10  ; #3腔电池破真空阀打开(A)
ANDLD
AND T0433  ; #3氦检原位延时确认
SET 12.14  ; #3电池破真空阀
LD TR0
LD 149.11  ; #3腔电池破真空阀关闭(M)
LD 1249.11  ; #3腔电池破真空阀关闭(A)
AND H0.01  ; 自动模式
ORLD
ANDLD
RSET 12.14  ; #3电池破真空阀

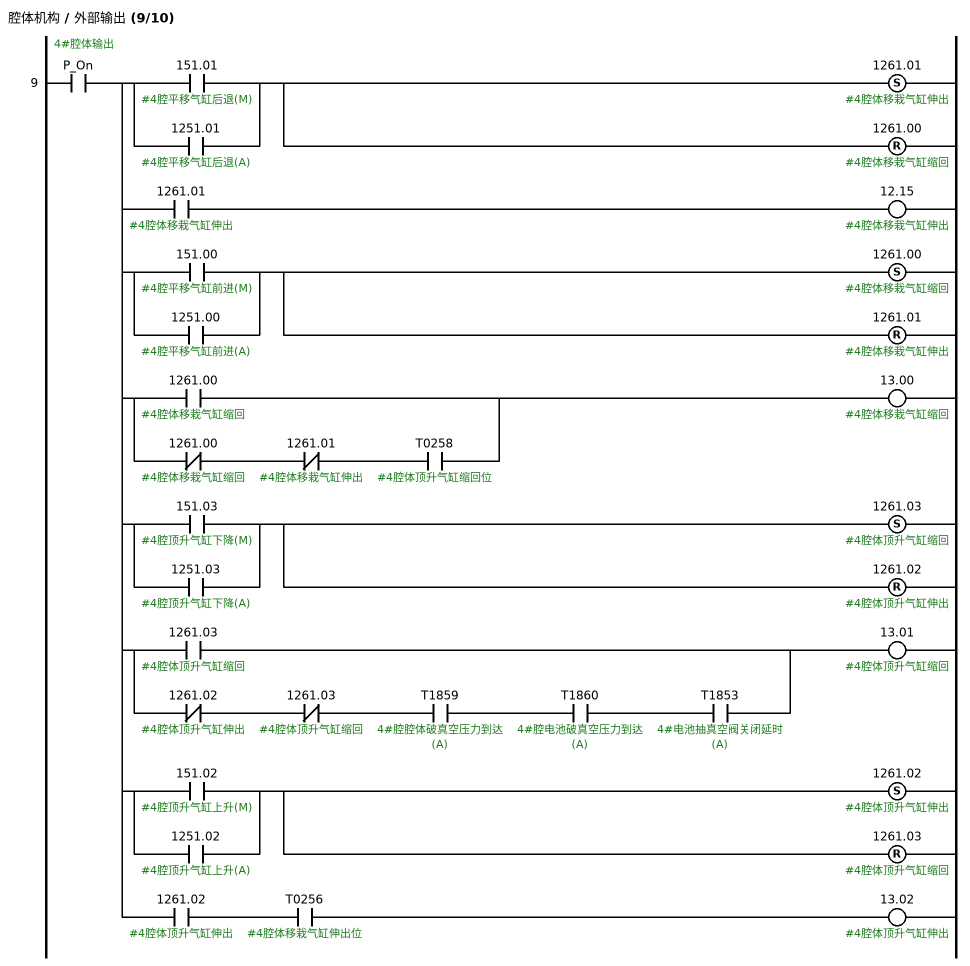
; rung 9: 4#腔体输出
LD P_On
OUT TR0
LD 151.01  ; #4腔平移气缸后退(M)
OR 1251.01  ; #4腔平移气缸后退(A)
ANDLD
SET 1261.01  ; #4腔体移栽气缸伸出
RSET 1261.00  ; #4腔体移栽气缸缩回
LD TR0
AND 1261.01  ; #4腔体移栽气缸伸出
OUT 12.15  ; #4腔体移栽气缸伸出
LD TR0
LD 151.00  ; #4腔平移气缸前进(M)
OR 1251.00  ; #4腔平移气缸前进(A)
ANDLD
SET 1261.00  ; #4腔体移栽气缸缩回
RSET 1261.01  ; #4腔体移栽气缸伸出
LD TR0
LD 1261.00  ; #4腔体移栽气缸缩回
LDNOT 1261.00  ; #4腔体移栽气缸缩回
ANDNOT 1261.01  ; #4腔体移栽气缸伸出
AND T0258  ; #4腔体顶升气缸缩回位
ORLD
ANDLD
OUT 13.00  ; #4腔体移栽气缸缩回
LD TR0
LD 151.03  ; #4腔顶升气缸下降(M)
OR 1251.03  ; #4腔顶升气缸下降(A)
ANDLD
SET 1261.03  ; #4腔体顶升气缸缩回
RSET 1261.02  ; #4腔体顶升气缸伸出
LD TR0
LD 1261.03  ; #4腔体顶升气缸缩回
LDNOT 1261.02  ; #4腔体顶升气缸伸出
ANDNOT 1261.03  ; #4腔体顶升气缸缩回
AND T1859  ; 4#腔腔体破真空压力到达(A)
AND T1860  ; 4#腔电池破真空压力到达(A)
AND T1853  ; 4#电池抽真空阀关闭延时(A)
ORLD
ANDLD
OUT 13.01  ; #4腔体顶升气缸缩回
LD TR0
LD 151.02  ; #4腔顶升气缸上升(M)
OR 1251.02  ; #4腔顶升气缸上升(A)
ANDLD
SET 1261.02  ; #4腔体顶升气缸伸出
RSET 1261.03  ; #4腔体顶升气缸缩回
LD TR0
AND 1261.02  ; #4腔体顶升气缸伸出
AND T0256  ; #4腔体移栽气缸伸出位
OUT 13.02  ; #4腔体顶升气缸伸出

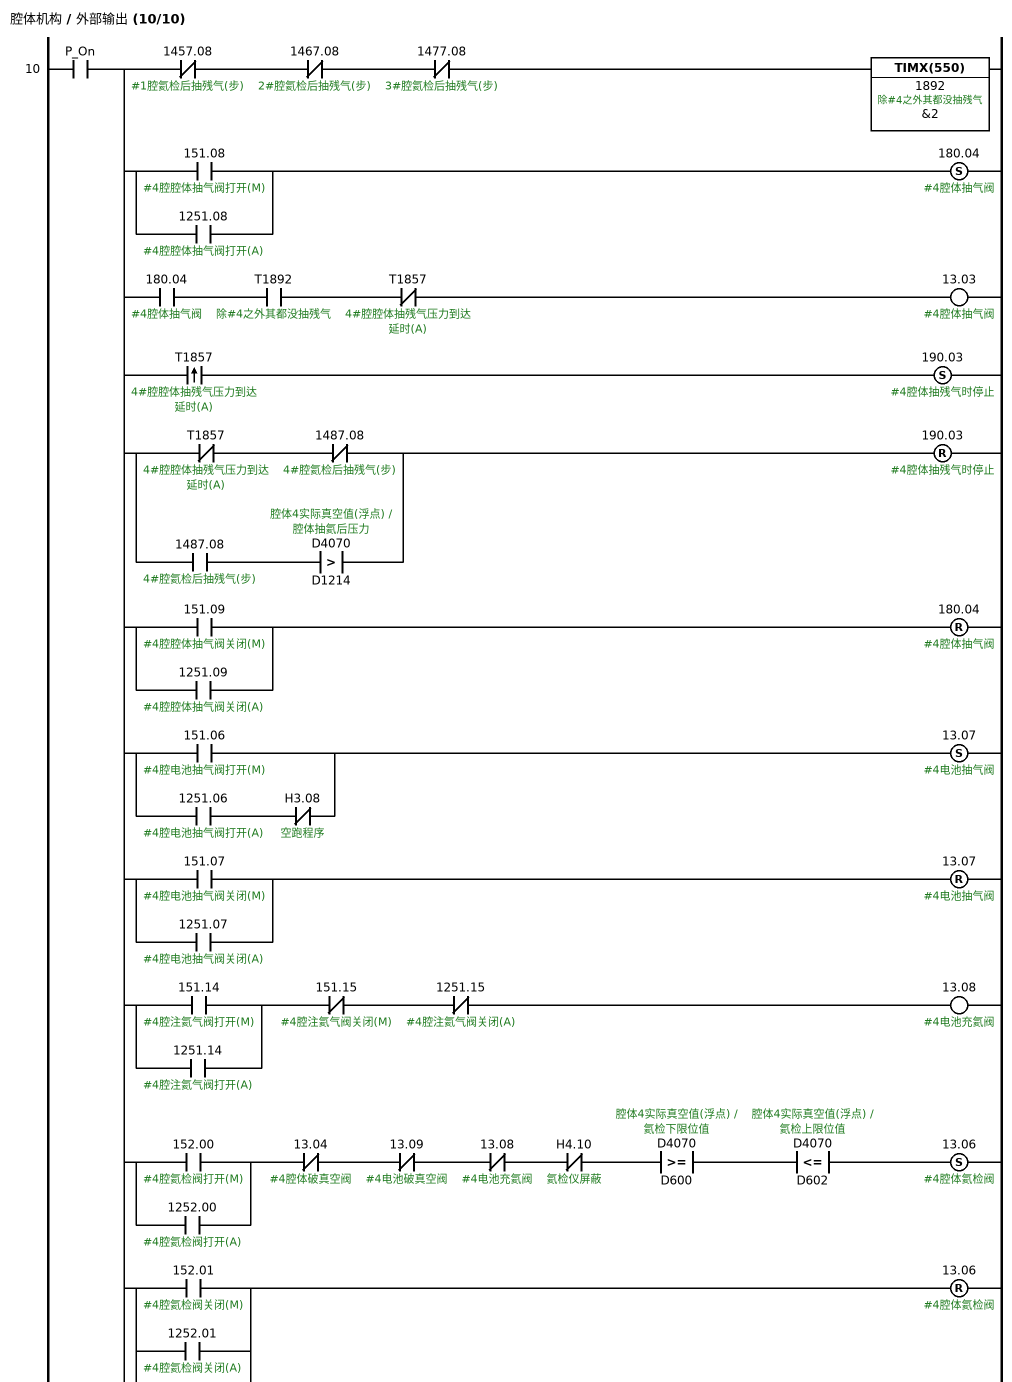

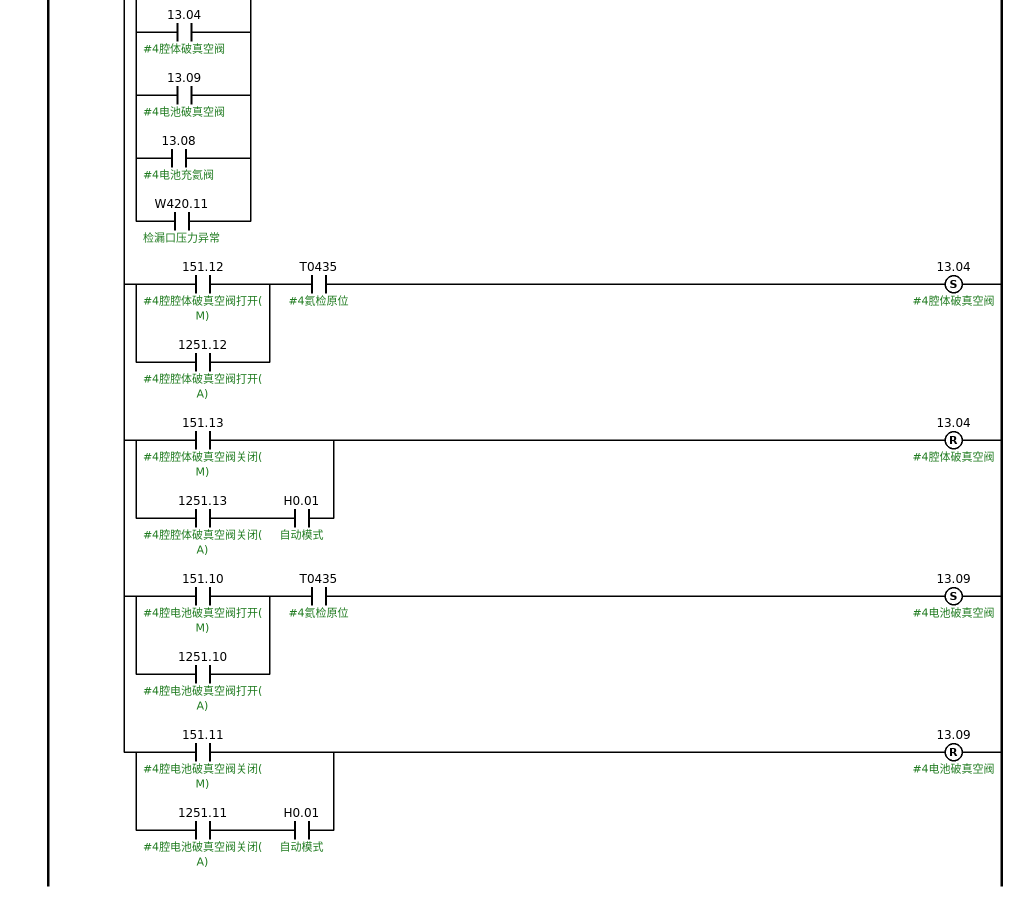
; rung 10
LD P_On
OUT TR0
ANDNOT 1457.08  ; #1腔氦检后抽残气(步)
ANDNOT 1467.08  ; 2#腔氦检后抽残气(步)
ANDNOT 1477.08  ; 3#腔氦检后抽残气(步)
TIMX(550) 1892 &2  ; 除#4之外其都没抽残气
LD TR0
LD 151.08  ; #4腔腔体抽气阀打开(M)
OR 1251.08  ; #4腔腔体抽气阀打开(A)
ANDLD
SET 180.04  ; #4腔体抽气阀
LD TR0
AND 180.04  ; #4腔体抽气阀
AND T1892  ; 除#4之外其都没抽残气
ANDNOT T1857  ; 4#腔腔体抽残气压力到达延时(A)
OUT 13.03  ; #4腔体抽气阀
LD TR0
@AND T1857  ; 4#腔腔体抽残气压力到达延时(A)
SET 190.03  ; #4腔体抽残气时停止
LD TR0
LDNOT T1857  ; 4#腔腔体抽残气压力到达延时(A)
ANDNOT 1487.08  ; 4#腔氦检后抽残气(步)
LD 1487.08  ; 4#腔氦检后抽残气(步)
AND>F(333) D4070 D1214  ; 腔体4实际真空值(浮点), 腔体抽氦后压力
ORLD
ANDLD
RSET 190.03  ; #4腔体抽残气时停止
LD TR0
LD 151.09  ; #4腔腔体抽气阀关闭(M)
OR 1251.09  ; #4腔腔体抽气阀关闭(A)
ANDLD
RSET 180.04  ; #4腔体抽气阀
LD TR0
LD 151.06  ; #4腔电池抽气阀打开(M)
LD 1251.06  ; #4腔电池抽气阀打开(A)
ANDNOT H3.08  ; 空跑程序
ORLD
ANDLD
SET 13.07  ; #4电池抽气阀
LD TR0
LD 151.07  ; #4腔电池抽气阀关闭(M)
OR 1251.07  ; #4腔电池抽气阀关闭(A)
ANDLD
RSET 13.07  ; #4电池抽气阀
LD TR0
LD 151.14  ; #4腔注氦气阀打开(M)
OR 1251.14  ; #4腔注氦气阀打开(A)
ANDLD
ANDNOT 151.15  ; #4腔注氦气阀关闭(M)
ANDNOT 1251.15  ; #4腔注氦气阀关闭(A)
OUT 13.08  ; #4电池充氦阀
LD TR0
LD 152.00  ; #4腔氦检阀打开(M)
OR 1252.00  ; #4腔氦检阀打开(A)
ANDLD
ANDNOT 13.04  ; #4腔体破真空阀
ANDNOT 13.09  ; #4电池破真空阀
ANDNOT 13.08  ; #4电池充氦阀
ANDNOT H4.10  ; 氦检仪屏蔽
AND>=F(334) D4070 D600  ; 腔体4实际真空值(浮点), 氦检下限位值
AND<=F(332) D4070 D602  ; 腔体4实际真空值(浮点), 氦检上限位值
SET 13.06  ; #4腔体氦检阀
LD TR0
LD 152.01  ; #4腔氦检阀关闭(M)
OR 1252.01  ; #4腔氦检阀关闭(A)
OR 13.04  ; #4腔体破真空阀
OR 13.09  ; #4电池破真空阀
OR 13.08  ; #4电池充氦阀
OR W420.11  ; 检漏口压力异常
ANDLD
RSET 13.06  ; #4腔体氦检阀
LD TR0
LD 151.12  ; #4腔腔体破真空阀打开(M)
OR 1251.12  ; #4腔腔体破真空阀打开(A)
ANDLD
AND T0435  ; #4氦检原位
SET 13.04  ; #4腔体破真空阀
LD TR0
LD 151.13  ; #4腔腔体破真空阀关闭(M)
LD 1251.13  ; #4腔腔体破真空阀关闭(A)
AND H0.01  ; 自动模式
ORLD
ANDLD
RSET 13.04  ; #4腔体破真空阀
LD TR0
LD 151.10  ; #4腔电池破真空阀打开(M)
OR 1251.10  ; #4腔电池破真空阀打开(A)
ANDLD
AND T0435  ; #4氦检原位
SET 13.09  ; #4电池破真空阀
LD TR0
LD 151.11  ; #4腔电池破真空阀关闭(M)
LD 1251.11  ; #4腔电池破真空阀关闭(A)
AND H0.01  ; 自动模式
ORLD
ANDLD
RSET 13.09  ; #4电池破真空阀

### Section 指示灯

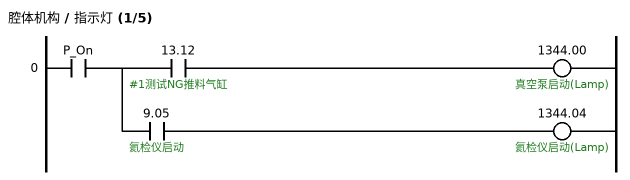
; rung 0
LD P_On
OUT TR0
AND 13.12  ; #1测试NG推料气缸
OUT 1344.00  ; 真空泵启动(Lamp)
LD TR0
AND 9.05  ; 氦检仪启动
OUT 1344.04  ; 氦检仪启动(Lamp)

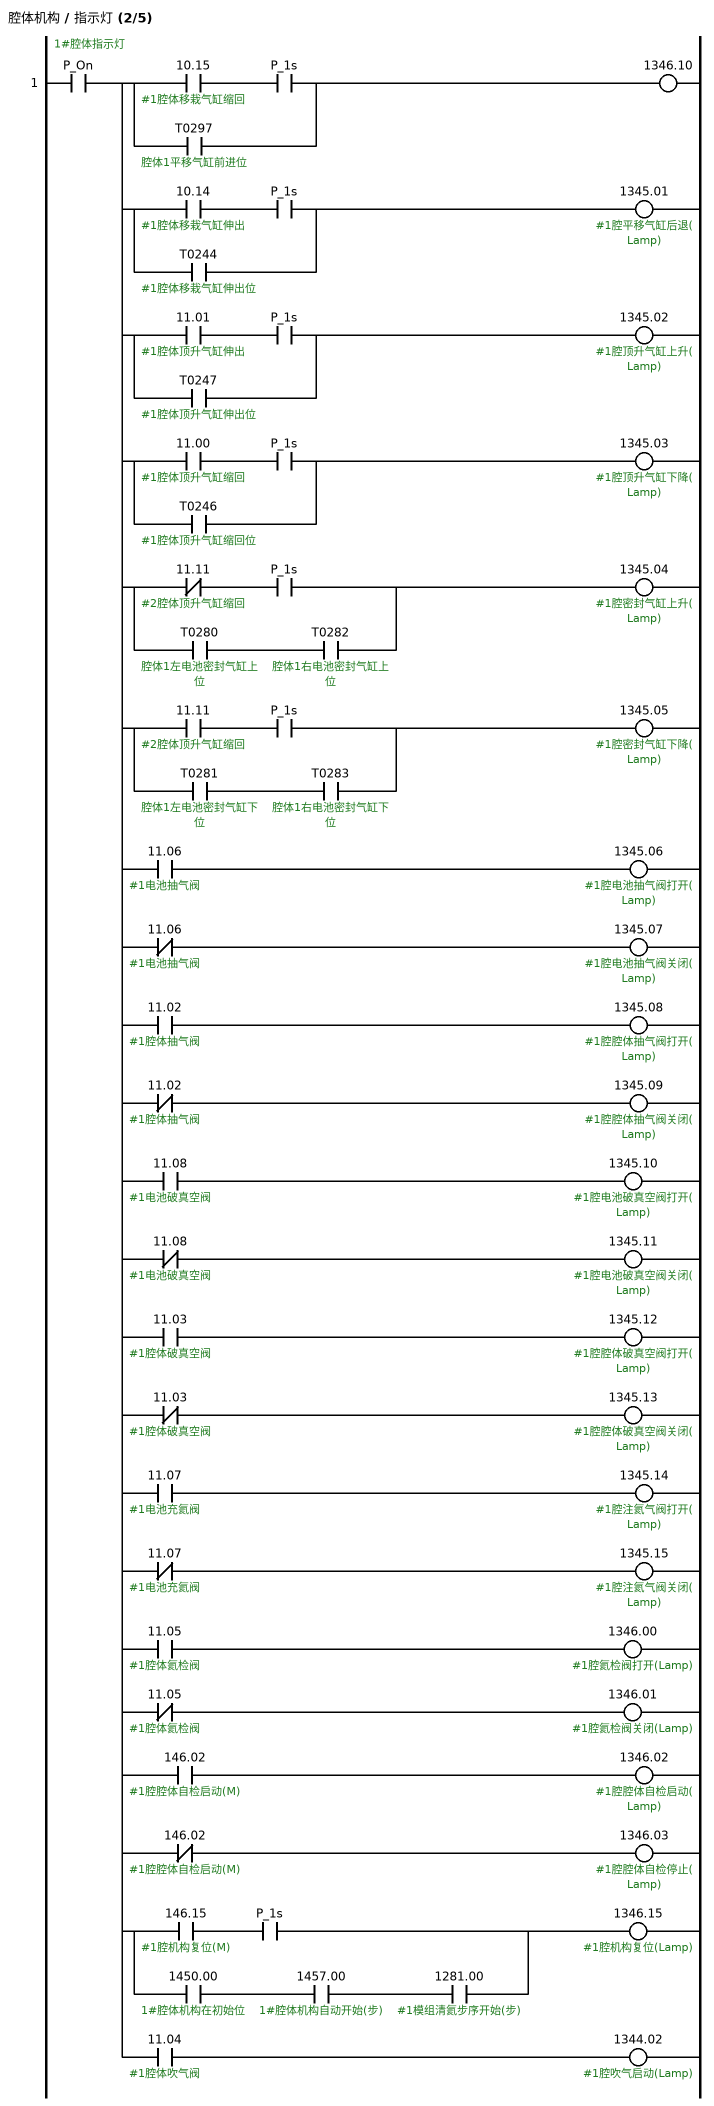
; rung 1: 1#腔体指示灯
LD P_On
OUT TR0
LD 10.15  ; #1腔体移栽气缸缩回
AND P_1s
OR T0297  ; 腔体1平移气缸前进位
ANDLD
OUT 1346.10
LD TR0
LD 10.14  ; #1腔体移栽气缸伸出
AND P_1s
OR T0244  ; #1腔体移栽气缸伸出位
ANDLD
OUT 1345.01  ; #1腔平移气缸后退(Lamp)
LD TR0
LD 11.01  ; #1腔体顶升气缸伸出
AND P_1s
OR T0247  ; #1腔体顶升气缸伸出位
ANDLD
OUT 1345.02  ; #1腔顶升气缸上升(Lamp)
LD TR0
LD 11.00  ; #1腔体顶升气缸缩回
AND P_1s
OR T0246  ; #1腔体顶升气缸缩回位
ANDLD
OUT 1345.03  ; #1腔顶升气缸下降(Lamp)
LD TR0
LDNOT 11.11  ; #2腔体顶升气缸缩回
AND P_1s
LD T0280  ; 腔体1左电池密封气缸上位
AND T0282  ; 腔体1右电池密封气缸上位
ORLD
ANDLD
OUT 1345.04  ; #1腔密封气缸上升(Lamp)
LD TR0
LD 11.11  ; #2腔体顶升气缸缩回
AND P_1s
LD T0281  ; 腔体1左电池密封气缸下位
AND T0283  ; 腔体1右电池密封气缸下位
ORLD
ANDLD
OUT 1345.05  ; #1腔密封气缸下降(Lamp)
LD TR0
AND 11.06  ; #1电池抽气阀
OUT 1345.06  ; #1腔电池抽气阀打开(Lamp)
LD TR0
ANDNOT 11.06  ; #1电池抽气阀
OUT 1345.07  ; #1腔电池抽气阀关闭(Lamp)
LD TR0
AND 11.02  ; #1腔体抽气阀
OUT 1345.08  ; #1腔腔体抽气阀打开(Lamp)
LD TR0
ANDNOT 11.02  ; #1腔体抽气阀
OUT 1345.09  ; #1腔腔体抽气阀关闭(Lamp)
LD TR0
AND 11.08  ; #1电池破真空阀
OUT 1345.10  ; #1腔电池破真空阀打开(Lamp)
LD TR0
ANDNOT 11.08  ; #1电池破真空阀
OUT 1345.11  ; #1腔电池破真空阀关闭(Lamp)
LD TR0
AND 11.03  ; #1腔体破真空阀
OUT 1345.12  ; #1腔腔体破真空阀打开(Lamp)
LD TR0
ANDNOT 11.03  ; #1腔体破真空阀
OUT 1345.13  ; #1腔腔体破真空阀关闭(Lamp)
LD TR0
AND 11.07  ; #1电池充氦阀
OUT 1345.14  ; #1腔注氦气阀打开(Lamp)
LD TR0
ANDNOT 11.07  ; #1电池充氦阀
OUT 1345.15  ; #1腔注氦气阀关闭(Lamp)
LD TR0
AND 11.05  ; #1腔体氦检阀
OUT 1346.00  ; #1腔氦检阀打开(Lamp)
LD TR0
ANDNOT 11.05  ; #1腔体氦检阀
OUT 1346.01  ; #1腔氦检阀关闭(Lamp)
LD TR0
AND 146.02  ; #1腔腔体自检启动(M)
OUT 1346.02  ; #1腔腔体自检启动(Lamp)
LD TR0
ANDNOT 146.02  ; #1腔腔体自检启动(M)
OUT 1346.03  ; #1腔腔体自检停止(Lamp)
LD TR0
LD 146.15  ; #1腔机构复位(M)
AND P_1s
LD 1450.00  ; 1#腔体机构在初始位
AND 1457.00  ; 1#腔体机构自动开始(步)
AND 1281.00  ; #1模组清氦步序开始(步)
ORLD
ANDLD
OUT 1346.15  ; #1腔机构复位(Lamp)
LD TR0
AND 11.04  ; #1腔体吹气阀
OUT 1344.02  ; #1腔吹气启动(Lamp)

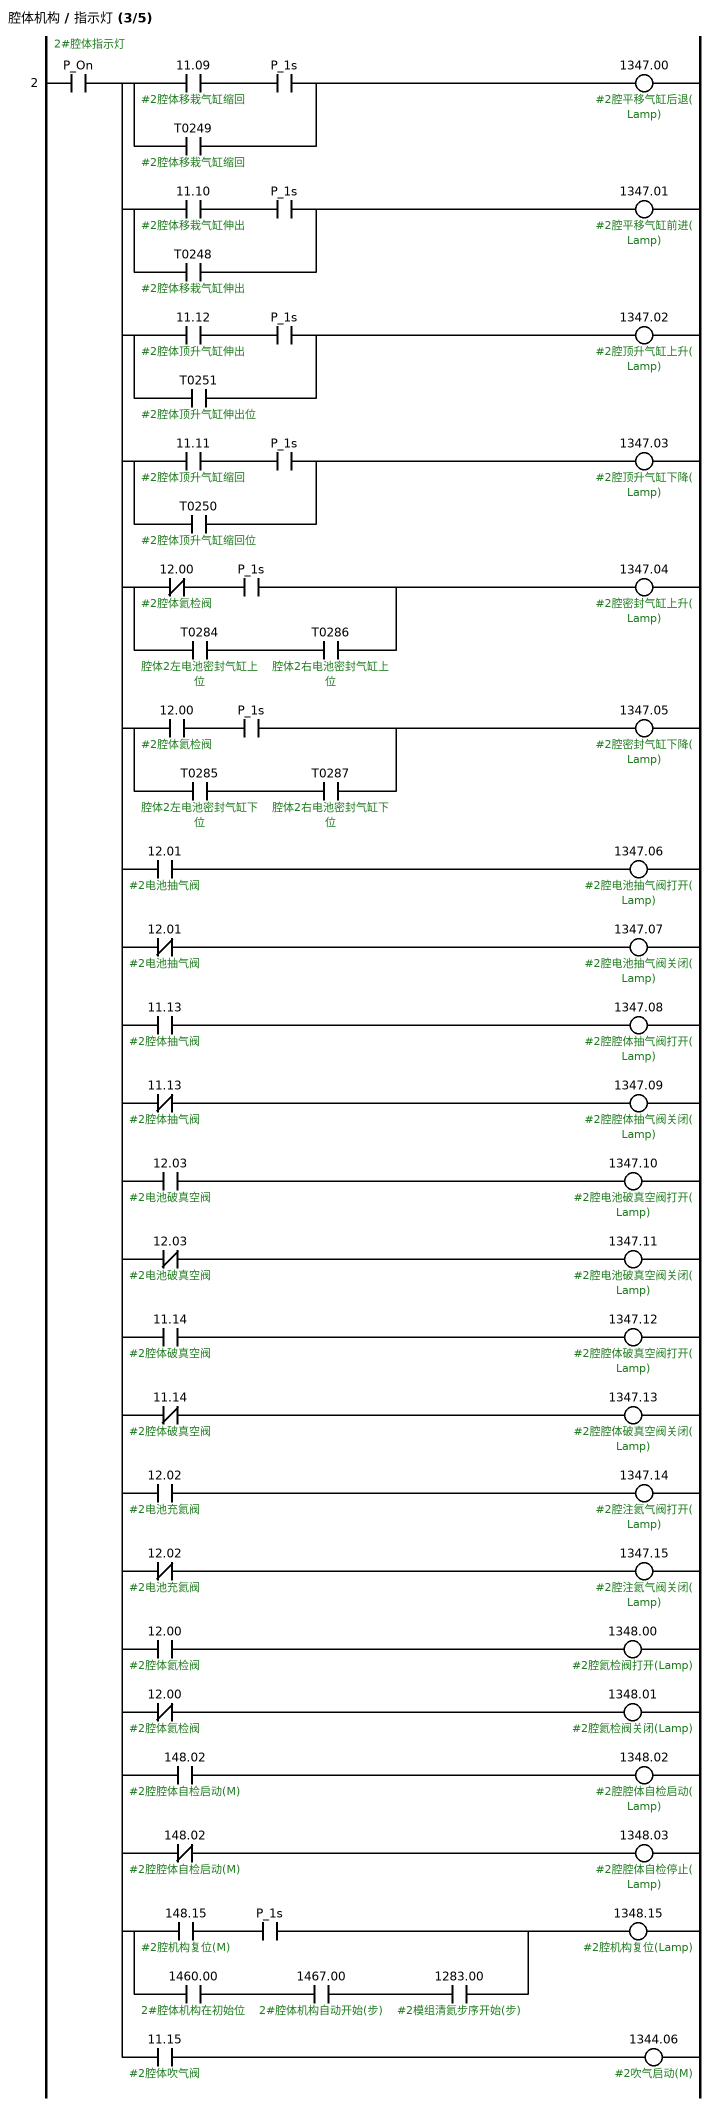
; rung 2: 2#腔体指示灯
LD P_On
OUT TR0
LD 11.09  ; #2腔体移栽气缸缩回
AND P_1s
OR T0249  ; #2腔体移栽气缸缩回
ANDLD
OUT 1347.00  ; #2腔平移气缸后退(Lamp)
LD TR0
LD 11.10  ; #2腔体移栽气缸伸出
AND P_1s
OR T0248  ; #2腔体移栽气缸伸出
ANDLD
OUT 1347.01  ; #2腔平移气缸前进(Lamp)
LD TR0
LD 11.12  ; #2腔体顶升气缸伸出
AND P_1s
OR T0251  ; #2腔体顶升气缸伸出位
ANDLD
OUT 1347.02  ; #2腔顶升气缸上升(Lamp)
LD TR0
LD 11.11  ; #2腔体顶升气缸缩回
AND P_1s
OR T0250  ; #2腔体顶升气缸缩回位
ANDLD
OUT 1347.03  ; #2腔顶升气缸下降(Lamp)
LD TR0
LDNOT 12.00  ; #2腔体氦检阀
AND P_1s
LD T0284  ; 腔体2左电池密封气缸上位
AND T0286  ; 腔体2右电池密封气缸上位
ORLD
ANDLD
OUT 1347.04  ; #2腔密封气缸上升(Lamp)
LD TR0
LD 12.00  ; #2腔体氦检阀
AND P_1s
LD T0285  ; 腔体2左电池密封气缸下位
AND T0287  ; 腔体2右电池密封气缸下位
ORLD
ANDLD
OUT 1347.05  ; #2腔密封气缸下降(Lamp)
LD TR0
AND 12.01  ; #2电池抽气阀
OUT 1347.06  ; #2腔电池抽气阀打开(Lamp)
LD TR0
ANDNOT 12.01  ; #2电池抽气阀
OUT 1347.07  ; #2腔电池抽气阀关闭(Lamp)
LD TR0
AND 11.13  ; #2腔体抽气阀
OUT 1347.08  ; #2腔腔体抽气阀打开(Lamp)
LD TR0
ANDNOT 11.13  ; #2腔体抽气阀
OUT 1347.09  ; #2腔腔体抽气阀关闭(Lamp)
LD TR0
AND 12.03  ; #2电池破真空阀
OUT 1347.10  ; #2腔电池破真空阀打开(Lamp)
LD TR0
ANDNOT 12.03  ; #2电池破真空阀
OUT 1347.11  ; #2腔电池破真空阀关闭(Lamp)
LD TR0
AND 11.14  ; #2腔体破真空阀
OUT 1347.12  ; #2腔腔体破真空阀打开(Lamp)
LD TR0
ANDNOT 11.14  ; #2腔体破真空阀
OUT 1347.13  ; #2腔腔体破真空阀关闭(Lamp)
LD TR0
AND 12.02  ; #2电池充氦阀
OUT 1347.14  ; #2腔注氦气阀打开(Lamp)
LD TR0
ANDNOT 12.02  ; #2电池充氦阀
OUT 1347.15  ; #2腔注氦气阀关闭(Lamp)
LD TR0
AND 12.00  ; #2腔体氦检阀
OUT 1348.00  ; #2腔氦检阀打开(Lamp)
LD TR0
ANDNOT 12.00  ; #2腔体氦检阀
OUT 1348.01  ; #2腔氦检阀关闭(Lamp)
LD TR0
AND 148.02  ; #2腔腔体自检启动(M)
OUT 1348.02  ; #2腔腔体自检启动(Lamp)
LD TR0
ANDNOT 148.02  ; #2腔腔体自检启动(M)
OUT 1348.03  ; #2腔腔体自检停止(Lamp)
LD TR0
LD 148.15  ; #2腔机构复位(M)
AND P_1s
LD 1460.00  ; 2#腔体机构在初始位
AND 1467.00  ; 2#腔体机构自动开始(步)
AND 1283.00  ; #2模组清氦步序开始(步)
ORLD
ANDLD
OUT 1348.15  ; #2腔机构复位(Lamp)
LD TR0
AND 11.15  ; #2腔体吹气阀
OUT 1344.06  ; #2吹气启动(M)

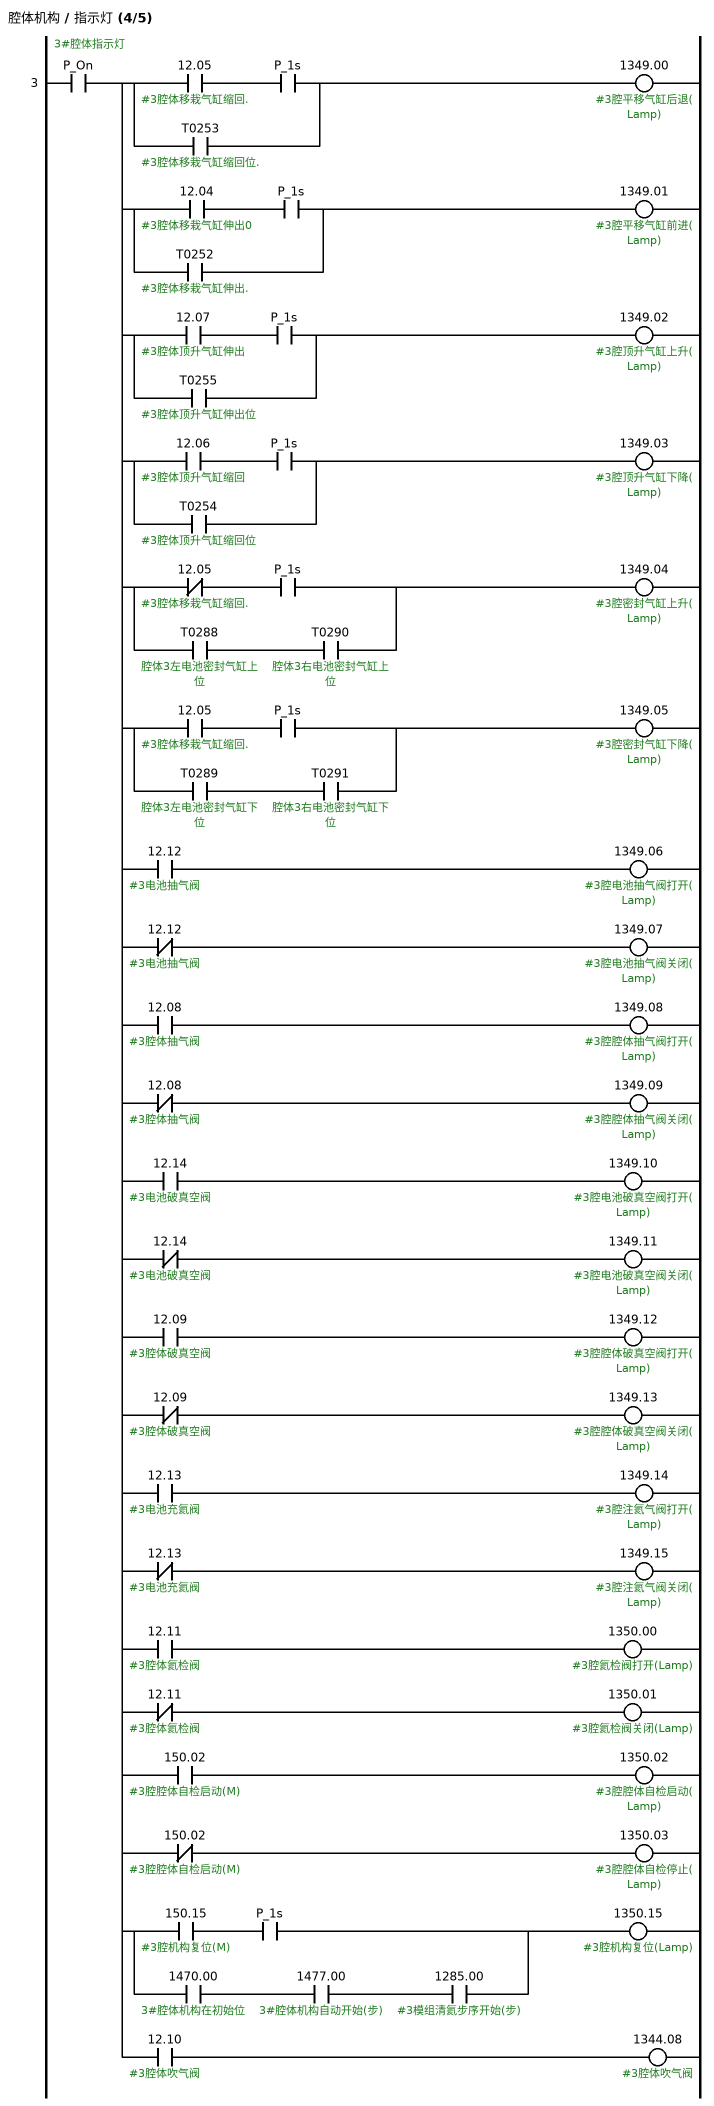
; rung 3: 3#腔体指示灯
LD P_On
OUT TR0
LD 12.05  ; #3腔体移栽气缸缩回.
AND P_1s
OR T0253  ; #3腔体移栽气缸缩回位.
ANDLD
OUT 1349.00  ; #3腔平移气缸后退(Lamp)
LD TR0
LD 12.04  ; #3腔体移栽气缸伸出0
AND P_1s
OR T0252  ; #3腔体移栽气缸伸出.
ANDLD
OUT 1349.01  ; #3腔平移气缸前进(Lamp)
LD TR0
LD 12.07  ; #3腔体顶升气缸伸出
AND P_1s
OR T0255  ; #3腔体顶升气缸伸出位
ANDLD
OUT 1349.02  ; #3腔顶升气缸上升(Lamp)
LD TR0
LD 12.06  ; #3腔体顶升气缸缩回
AND P_1s
OR T0254  ; #3腔体顶升气缸缩回位
ANDLD
OUT 1349.03  ; #3腔顶升气缸下降(Lamp)
LD TR0
LDNOT 12.05  ; #3腔体移栽气缸缩回.
AND P_1s
LD T0288  ; 腔体3左电池密封气缸上位
AND T0290  ; 腔体3右电池密封气缸上位
ORLD
ANDLD
OUT 1349.04  ; #3腔密封气缸上升(Lamp)
LD TR0
LD 12.05  ; #3腔体移栽气缸缩回.
AND P_1s
LD T0289  ; 腔体3左电池密封气缸下位
AND T0291  ; 腔体3右电池密封气缸下位
ORLD
ANDLD
OUT 1349.05  ; #3腔密封气缸下降(Lamp)
LD TR0
AND 12.12  ; #3电池抽气阀
OUT 1349.06  ; #3腔电池抽气阀打开(Lamp)
LD TR0
ANDNOT 12.12  ; #3电池抽气阀
OUT 1349.07  ; #3腔电池抽气阀关闭(Lamp)
LD TR0
AND 12.08  ; #3腔体抽气阀
OUT 1349.08  ; #3腔腔体抽气阀打开(Lamp)
LD TR0
ANDNOT 12.08  ; #3腔体抽气阀
OUT 1349.09  ; #3腔腔体抽气阀关闭(Lamp)
LD TR0
AND 12.14  ; #3电池破真空阀
OUT 1349.10  ; #3腔电池破真空阀打开(Lamp)
LD TR0
ANDNOT 12.14  ; #3电池破真空阀
OUT 1349.11  ; #3腔电池破真空阀关闭(Lamp)
LD TR0
AND 12.09  ; #3腔体破真空阀
OUT 1349.12  ; #3腔腔体破真空阀打开(Lamp)
LD TR0
ANDNOT 12.09  ; #3腔体破真空阀
OUT 1349.13  ; #3腔腔体破真空阀关闭(Lamp)
LD TR0
AND 12.13  ; #3电池充氦阀
OUT 1349.14  ; #3腔注氦气阀打开(Lamp)
LD TR0
ANDNOT 12.13  ; #3电池充氦阀
OUT 1349.15  ; #3腔注氦气阀关闭(Lamp)
LD TR0
AND 12.11  ; #3腔体氦检阀
OUT 1350.00  ; #3腔氦检阀打开(Lamp)
LD TR0
ANDNOT 12.11  ; #3腔体氦检阀
OUT 1350.01  ; #3腔氦检阀关闭(Lamp)
LD TR0
AND 150.02  ; #3腔腔体自检启动(M)
OUT 1350.02  ; #3腔腔体自检启动(Lamp)
LD TR0
ANDNOT 150.02  ; #3腔腔体自检启动(M)
OUT 1350.03  ; #3腔腔体自检停止(Lamp)
LD TR0
LD 150.15  ; #3腔机构复位(M)
AND P_1s
LD 1470.00  ; 3#腔体机构在初始位
AND 1477.00  ; 3#腔体机构自动开始(步)
AND 1285.00  ; #3模组清氦步序开始(步)
ORLD
ANDLD
OUT 1350.15  ; #3腔机构复位(Lamp)
LD TR0
AND 12.10  ; #3腔体吹气阀
OUT 1344.08  ; #3腔体吹气阀

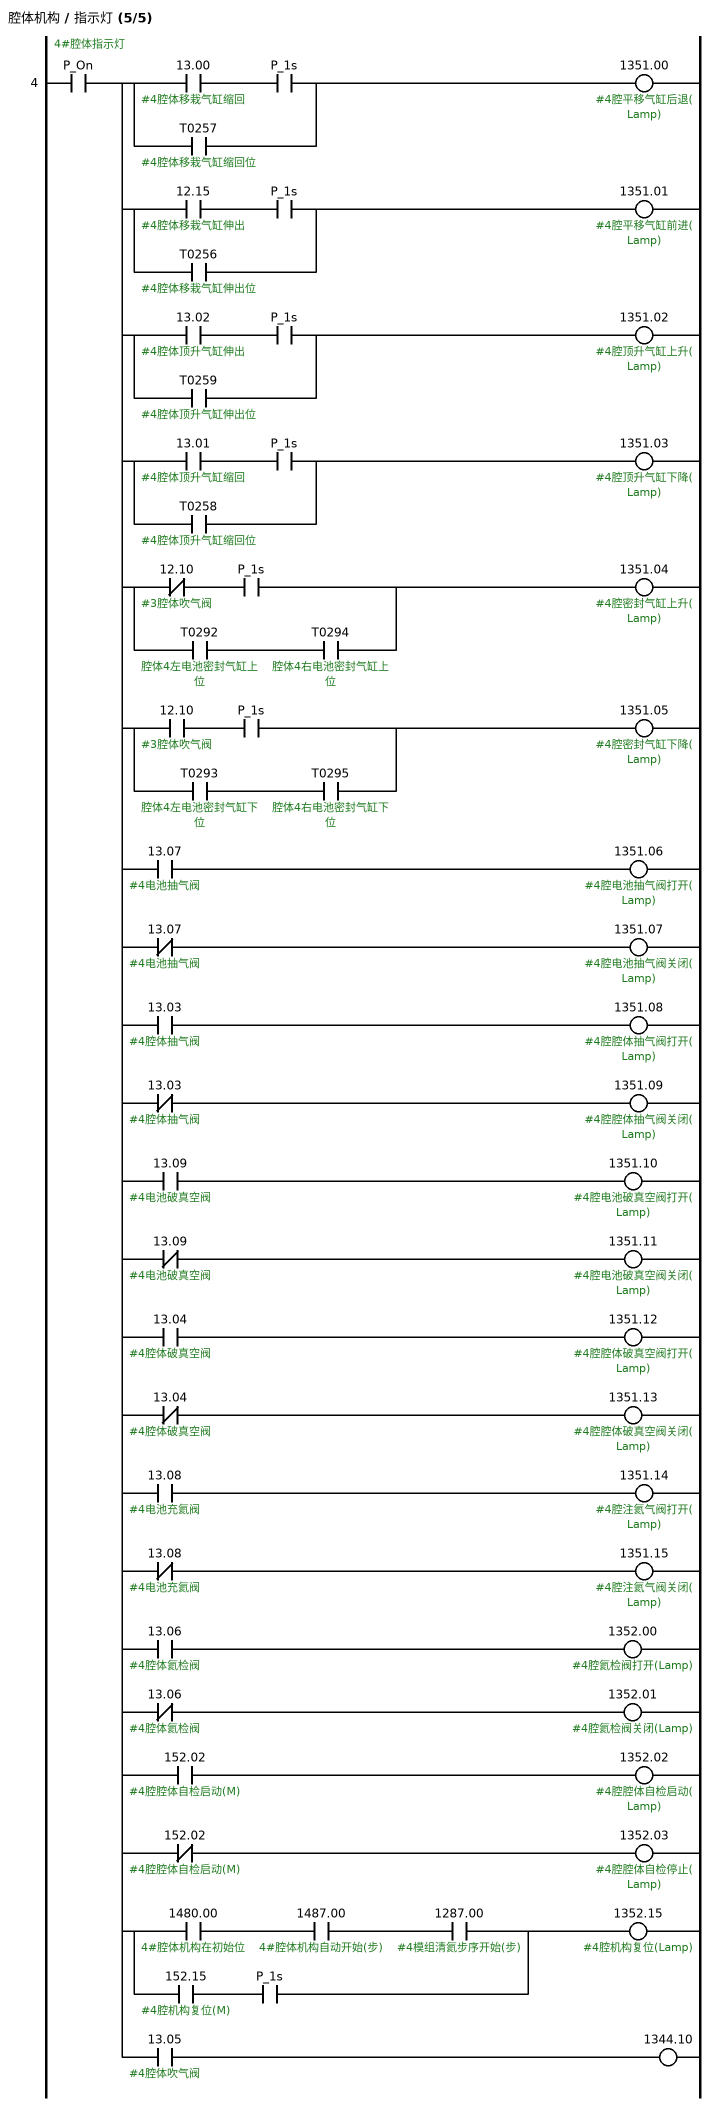
; rung 4: 4#腔体指示灯
LD P_On
OUT TR0
LD 13.00  ; #4腔体移栽气缸缩回
AND P_1s
OR T0257  ; #4腔体移栽气缸缩回位
ANDLD
OUT 1351.00  ; #4腔平移气缸后退(Lamp)
LD TR0
LD 12.15  ; #4腔体移栽气缸伸出
AND P_1s
OR T0256  ; #4腔体移栽气缸伸出位
ANDLD
OUT 1351.01  ; #4腔平移气缸前进(Lamp)
LD TR0
LD 13.02  ; #4腔体顶升气缸伸出
AND P_1s
OR T0259  ; #4腔体顶升气缸伸出位
ANDLD
OUT 1351.02  ; #4腔顶升气缸上升(Lamp)
LD TR0
LD 13.01  ; #4腔体顶升气缸缩回
AND P_1s
OR T0258  ; #4腔体顶升气缸缩回位
ANDLD
OUT 1351.03  ; #4腔顶升气缸下降(Lamp)
LD TR0
LDNOT 12.10  ; #3腔体吹气阀
AND P_1s
LD T0292  ; 腔体4左电池密封气缸上位
AND T0294  ; 腔体4右电池密封气缸上位
ORLD
ANDLD
OUT 1351.04  ; #4腔密封气缸上升(Lamp)
LD TR0
LD 12.10  ; #3腔体吹气阀
AND P_1s
LD T0293  ; 腔体4左电池密封气缸下位
AND T0295  ; 腔体4右电池密封气缸下位
ORLD
ANDLD
OUT 1351.05  ; #4腔密封气缸下降(Lamp)
LD TR0
AND 13.07  ; #4电池抽气阀
OUT 1351.06  ; #4腔电池抽气阀打开(Lamp)
LD TR0
ANDNOT 13.07  ; #4电池抽气阀
OUT 1351.07  ; #4腔电池抽气阀关闭(Lamp)
LD TR0
AND 13.03  ; #4腔体抽气阀
OUT 1351.08  ; #4腔腔体抽气阀打开(Lamp)
LD TR0
ANDNOT 13.03  ; #4腔体抽气阀
OUT 1351.09  ; #4腔腔体抽气阀关闭(Lamp)
LD TR0
AND 13.09  ; #4电池破真空阀
OUT 1351.10  ; #4腔电池破真空阀打开(Lamp)
LD TR0
ANDNOT 13.09  ; #4电池破真空阀
OUT 1351.11  ; #4腔电池破真空阀关闭(Lamp)
LD TR0
AND 13.04  ; #4腔体破真空阀
OUT 1351.12  ; #4腔腔体破真空阀打开(Lamp)
LD TR0
ANDNOT 13.04  ; #4腔体破真空阀
OUT 1351.13  ; #4腔腔体破真空阀关闭(Lamp)
LD TR0
AND 13.08  ; #4电池充氦阀
OUT 1351.14  ; #4腔注氦气阀打开(Lamp)
LD TR0
ANDNOT 13.08  ; #4电池充氦阀
OUT 1351.15  ; #4腔注氦气阀关闭(Lamp)
LD TR0
AND 13.06  ; #4腔体氦检阀
OUT 1352.00  ; #4腔氦检阀打开(Lamp)
LD TR0
ANDNOT 13.06  ; #4腔体氦检阀
OUT 1352.01  ; #4腔氦检阀关闭(Lamp)
LD TR0
AND 152.02  ; #4腔腔体自检启动(M)
OUT 1352.02  ; #4腔腔体自检启动(Lamp)
LD TR0
ANDNOT 152.02  ; #4腔腔体自检启动(M)
OUT 1352.03  ; #4腔腔体自检停止(Lamp)
LD TR0
LD 1480.00  ; 4#腔体机构在初始位
AND 1487.00  ; 4#腔体机构自动开始(步)
AND 1287.00  ; #4模组清氦步序开始(步)
LD 152.15  ; #4腔机构复位(M)
AND P_1s
ORLD
ANDLD
OUT 1352.15  ; #4腔机构复位(Lamp)
LD TR0
AND 13.05  ; #4腔体吹气阀
OUT 1344.10

### Section END
; rung 0
END(001)

## Program COMMON (cyclic task 7)
Local symbols
ccf113 BOOL

### Section Main

### Section 延时

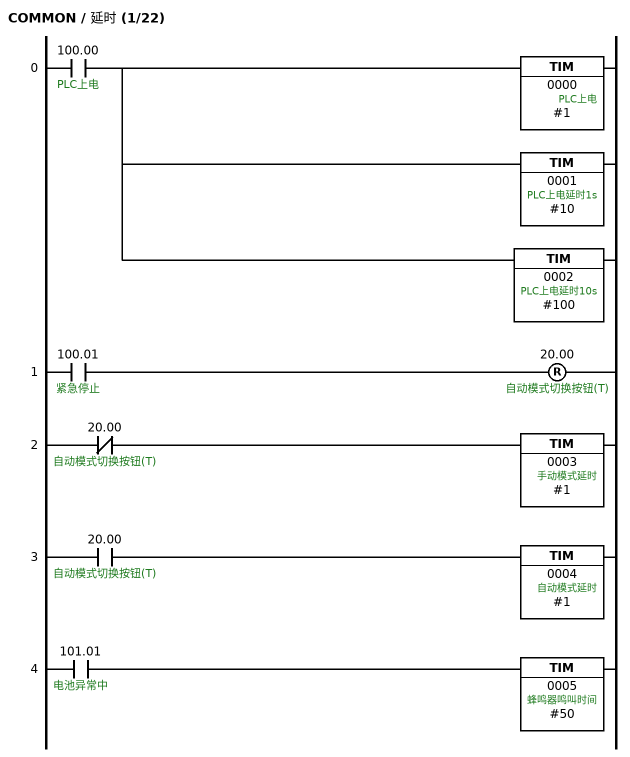
; rung 0
LD 100.00  ; PLC上电
TIM 0000 #1  ; PLC上电
TIM 0001 #10  ; PLC上电延时1s
TIM 0002 #100  ; PLC上电延时10s
; rung 1
LD 100.01  ; 紧急停止
RSET 20.00  ; 自动模式切换按钮(T)
; rung 2
LDNOT 20.00  ; 自动模式切换按钮(T)
TIM 0003 #1  ; 手动模式延时
; rung 3
LD 20.00  ; 自动模式切换按钮(T)
TIM 0004 #1  ; 自动模式延时
; rung 4
LD 101.01  ; 电池异常中
TIM 0005 #50  ; 蜂鸣器鸣叫时间

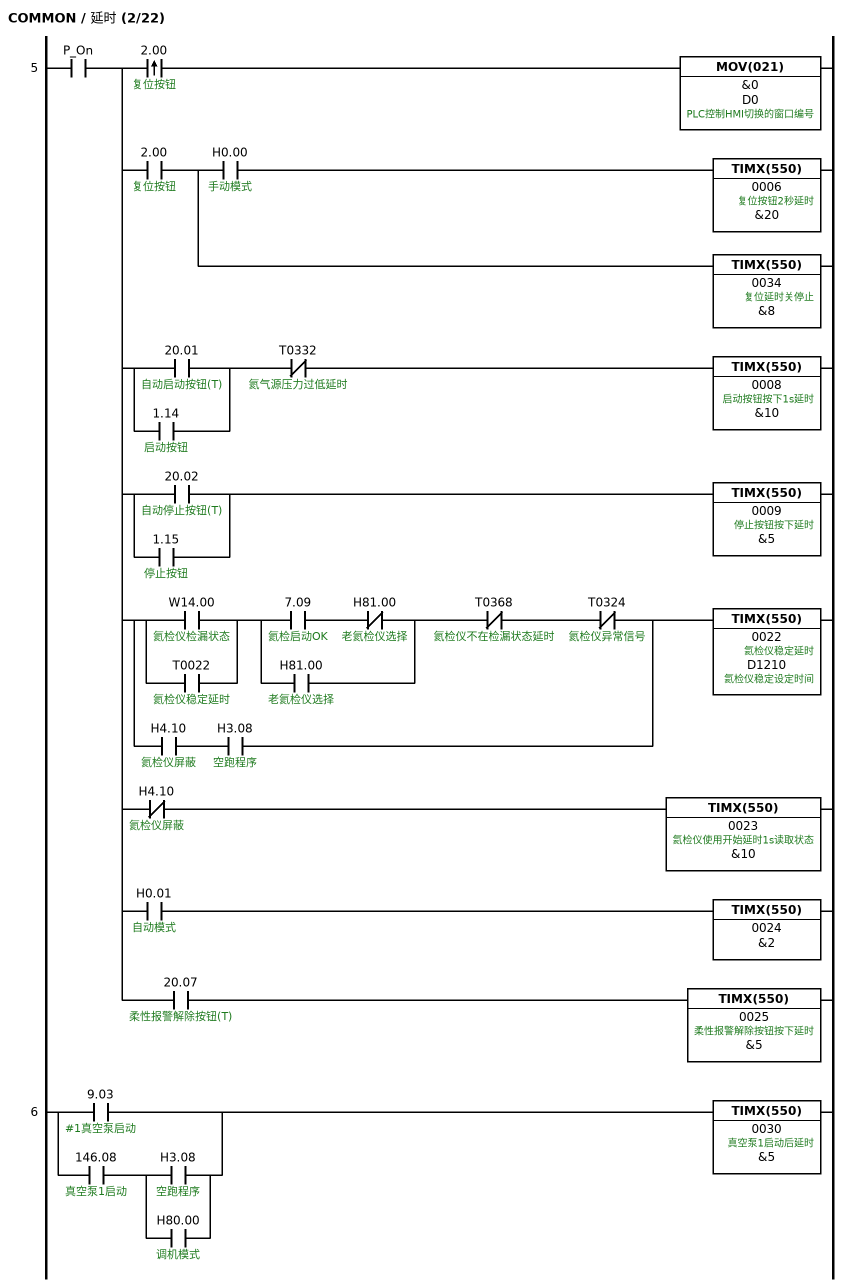
; rung 5
LD P_On
OUT TR0
@AND 2.00  ; 复位按钮
MOV(021) &0 D0  ; PLC控制HMI切换的窗口编号
LD TR0
AND 2.00  ; 复位按钮
OUT TR1
AND H0.00  ; 手动模式
TIMX(550) 0006 &20  ; 复位按钮2秒延时
LD TR1
TIMX(550) 0034 &8  ; 复位延时关停止
LD TR0
LD 20.01  ; 自动启动按钮(T)
OR 1.14  ; 启动按钮
ANDLD
ANDNOT T0332  ; 氦气源压力过低延时
TIMX(550) 0008 &10  ; 启动按钮按下1s延时
LD TR0
LD 20.02  ; 自动停止按钮(T)
OR 1.15  ; 停止按钮
ANDLD
TIMX(550) 0009 &5  ; 停止按钮按下延时
LD TR0
LD W14.00  ; 氦检仪检漏状态
OR T0022  ; 氦检仪稳定延时
LD 7.09  ; 氦检启动OK
ANDNOT H81.00  ; 老氦检仪选择
OR H81.00  ; 老氦检仪选择
ANDLD
ANDNOT T0368  ; 氦检仪不在检漏状态延时
ANDNOT T0324  ; 氦检仪异常信号
LD H4.10  ; 氦检仪屏蔽
AND H3.08  ; 空跑程序
ORLD
ANDLD
TIMX(550) 0022 D1210  ; 氦检仪稳定设定时间, 氦检仪稳定延时
LD TR0
ANDNOT H4.10  ; 氦检仪屏蔽
TIMX(550) 0023 &10  ; 氦检仪使用开始延时1s读取状态
LD TR0
AND H0.01  ; 自动模式
TIMX(550) 0024 &2
LD TR0
AND 20.07  ; 柔性报警解除按钮(T)
TIMX(550) 0025 &5  ; 柔性报警解除按钮按下延时
; rung 6
LD 9.03  ; #1真空泵启动
LD 146.08  ; 真空泵1启动
LD H3.08  ; 空跑程序
OR H80.00  ; 调机模式
ANDLD
ORLD
TIMX(550) 0030 &5  ; 真空泵1启动后延时

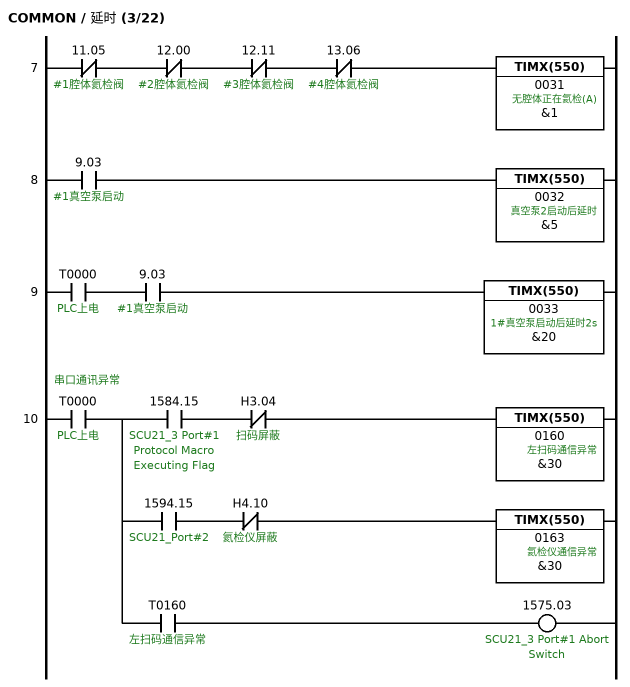
; rung 7
LDNOT 11.05  ; #1腔体氦检阀
ANDNOT 12.00  ; #2腔体氦检阀
ANDNOT 12.11  ; #3腔体氦检阀
ANDNOT 13.06  ; #4腔体氦检阀
TIMX(550) 0031 &1  ; 无腔体正在氦检(A)
; rung 8
LD 9.03  ; #1真空泵启动
TIMX(550) 0032 &5  ; 真空泵2启动后延时
; rung 9
LD T0000  ; PLC上电
AND 9.03  ; #1真空泵启动
TIMX(550) 0033 &20  ; 1#真空泵启动后延时2s
; rung 10: 串口通讯异常
LD T0000  ; PLC上电
OUT TR0
AND 1584.15  ; SCU21_3 Port#1 Protocol Macro Executing Flag
ANDNOT H3.04  ; 扫码屏蔽
TIMX(550) 0160 &30  ; 左扫码通信异常
LD TR0
AND 1594.15  ; SCU21_Port#2
ANDNOT H4.10  ; 氦检仪屏蔽
TIMX(550) 0163 &30  ; 氦检仪通信异常
LD TR0
AND T0160  ; 左扫码通信异常
OUT 1575.03  ; SCU21_3 Port#1 Abort Switch

